LIN {X 0.048,Y -151.819,Z 1203.251,A 0.000,B 0.000,C 90.000,E1 225.162} C_DIS
LIN {X 0.060,Y -150.032,Z 1203.236,A 0.000,B 0.000,C 90.000,E1 222.447} C_DIS
LIN {X -0.026,Y -146.851,Z 1203.211,A 0.000,B 0.000,C 90.000,E1 217.935} C_DIS
LIN {X -0.008,Y -145.434,Z 1203.195,A 0.000,B 0.000,C 90.000,E1 215.185} C_DIS
LIN {X -0.012,Y -142.857,Z 1203.170,A 0.000,B 0.000,C 90.000,E1 210.590} C_DIS
LIN {X 0.040,Y -141.472,Z 1203.149,A 0.000,B 0.000,C 90.000,E1 206.873} C_DIS
LIN {X 0.031,Y -139.379,Z 1203.113,A 0.000,B 0.000,C 90.000,E1 200.375} C_DIS
LIN {X 0.021,Y -138.831,Z 1203.098,A 0.000,B 0.000,C 90.000,E1 197.583} C_DIS
LIN {X -0.051,Y -138.353,Z 1203.056,A 0.000,B 0.000,C 90.000,E1 190.141} C_DIS
LIN {X -0.056,Y -139.527,Z 1203.004,A 0.000,B 0.000,C 90.000,E1 180.802} C_DIS
LIN {X 0.036,Y -141.198,Z 1202.973,A 0.000,B 0.000,C 90.000,E1 175.179} C_DIS
LIN {X -0.005,Y -142.575,Z 1202.958,A 0.000,B 0.000,C 90.000,E1 172.413} C_DIS
LIN {X -0.050,Y -144.865,Z 1202.932,A 0.000,B 0.000,C 90.000,E1 167.813} C_DIS
LIN {X 0.047,Y -147.491,Z 1202.912,A 0.000,B 0.000,C 90.000,E1 164.102} C_DIS
LIN {X -0.019,Y -150.080,Z 1202.891,A 0.000,B 0.000,C 90.000,E1 160.477} C_DIS
LIN {X -0.006,Y -153.430,Z 1202.871,A 0.000,B 0.000,C 90.000,E1 156.847} C_DIS
LIN {X -0.018,Y -156.851,Z 1202.851,A 0.000,B 0.000,C 90.000,E1 153.256} C_DIS
LIN {X 0.053,Y -160.933,Z 1202.832,A 0.000,B 0.000,C 90.000,E1 149.665} C_DIS
LIN {X -0.004,Y -163.056,Z 1202.822,A 0.000,B 0.000,C 90.000,E1 147.916} C_DIS
LIN {X 0.001,Y -167.451,Z 1202.802,A 0.000,B 0.000,C 90.000,E1 144.402} C_DIS
LIN {X -0.090,Y -171.289,Z 1202.788,A 0.000,B 0.000,C 90.000,E1 141.823} C_DIS
LIN {X 0.080,Y -176.182,Z 1202.769,A 0.000,B 0.000,C 90.000,E1 138.324} C_DIS
LIN {X -0.055,Y -180.457,Z 1202.754,A 0.000,B 0.000,C 90.000,E1 135.810} C_DIS
LIN {X -0.079,Y -185.862,Z 1202.736,A 0.000,B 0.000,C 90.000,E1 132.447} C_DIS
LIN {X -0.026,Y -190.485,Z 1202.722,A 0.000,B 0.000,C 90.000,E1 129.930} C_DIS
LIN {X -0.006,Y -196.237,Z 1202.703,A 0.000,B 0.000,C 90.000,E1 126.629} C_DIS
LIN {X 0.003,Y -201.371,Z 1202.689,A 0.000,B 0.000,C 90.000,E1 123.992} C_DIS
LIN {X 0.020,Y -201.579,Z 1202.688,A 0.000,B 0.000,C 90.000,E1 123.865} C_DIS
LIN {X -0.004,Y -311.934,Z 1202.688,A 0.000,B 0.000,C 90.000,E1 123.865} C_DIS
LIN {X -0.100,Y -314.414,Z 1202.688,A 0.000,B 0.000,C 90.000,E1 123.833} C_DIS
LIN {X 0.095,Y -318.650,Z 1202.687,A 0.000,B 0.000,C 90.000,E1 123.579} C_DIS
LIN {X 0.026,Y -321.137,Z 1202.685,A 0.000,B 0.000,C 90.000,E1 123.372} C_DIS
LIN {X -0.050,Y -324.912,Z 1202.683,A 0.000,B 0.000,C 90.000,E1 122.880} C_DIS
LIN {X 0.036,Y -326.560,Z 1202.681,A 0.000,B 0.000,C 90.000,E1 122.546} C_DIS
LIN {X -0.052,Y -333.737,Z 1202.670,A 0.000,B 0.000,C 90.000,E1 120.669} C_DIS
LIN {X 0.128,Y -345.390,Z 1202.655,A 0.000,B 0.000,C 90.000,E1 117.847} C_DIS
LIN {X -0.146,Y -358.479,Z 1202.640,A 0.000,B 0.000,C 90.000,E1 115.155} C_DIS
LIN {X -0.126,Y -371.413,Z 1202.626,A 0.000,B 0.000,C 90.000,E1 112.770} C_DIS
LIN {X -0.068,Y -385.665,Z 1202.613,A 0.000,B 0.000,C 90.000,E1 110.429} C_DIS
LIN {X 0.090,Y -401.333,Z 1202.601,A 0.000,B 0.000,C 90.000,E1 108.127} C_DIS
LIN {X 0.132,Y -418.530,Z 1202.588,A 0.000,B 0.000,C 90.000,E1 105.898} C_DIS
LIN {X -0.161,Y -437.373,Z 1202.576,A 0.000,B 0.000,C 90.000,E1 103.772} C_DIS
LIN {X -0.061,Y -457.365,Z 1202.565,A 0.000,B 0.000,C 90.000,E1 101.715} C_DIS
LIN {X 0.202,Y -470.159,Z 1202.558,A 0.000,B 0.000,C 90.000,E1 100.489} C_DIS
LIN {X -0.210,Y -472.456,Z 1202.557,A 0.000,B 0.000,C 90.000,E1 100.310} C_DIS
LIN {X -0.161,Y -474.191,Z 1202.556,A 0.000,B 0.000,C 90.000,E1 100.074} C_DIS
LIN {X 0.087,Y -475.642,Z 1202.554,A 0.000,B 0.000,C 90.000,E1 99.792} C_DIS
LIN {X -0.053,Y -476.723,Z 1202.553,A 0.000,B 0.000,C 90.000,E1 99.557} C_DIS
LIN {X 0.155,Y -477.992,Z 1202.550,A 0.000,B 0.000,C 90.000,E1 99.029} C_DIS
LIN {X -0.179,Y -478.247,Z 1202.547,A 0.000,B 0.000,C 90.000,E1 98.568} C_DIS
LIN {X -0.032,Y -477.531,Z 1202.545,A 0.000,B 0.000,C 90.000,E1 98.049} C_DIS
LIN {X 0.120,Y -475.728,Z 1202.542,A 0.000,B 0.000,C 90.000,E1 97.530} C_DIS
LIN {X -0.012,Y -474.315,Z 1202.541,A 0.000,B 0.000,C 90.000,E1 97.296} C_DIS
LIN {X 0.182,Y -457.953,Z 1202.528,A 0.000,B 0.000,C 90.000,E1 94.992} C_DIS
LIN {X 0.101,Y -440.459,Z 1202.513,A 0.000,B 0.000,C 90.000,E1 92.407} C_DIS
LIN {X 0.061,Y -422.849,Z 1202.497,A 0.000,B 0.000,C 90.000,E1 89.484} C_DIS
LIN {X 0.074,Y -411.058,Z 1202.485,A 0.000,B 0.000,C 90.000,E1 87.306} C_DIS
LIN {X -0.140,Y -399.438,Z 1202.473,A 0.000,B 0.000,C 90.000,E1 85.122} C_DIS
LIN {X 0.154,Y -389.245,Z 1202.462,A 0.000,B 0.000,C 90.000,E1 83.109} C_DIS
LIN {X -0.068,Y -378.977,Z 1202.451,A 0.000,B 0.000,C 90.000,E1 81.141} C_DIS
LIN {X -0.060,Y -369.917,Z 1202.441,A 0.000,B 0.000,C 90.000,E1 79.398} C_DIS
LIN {X -0.178,Y -358.952,Z 1202.430,A 0.000,B 0.000,C 90.000,E1 77.353} C_DIS
LIN {X -0.028,Y -347.727,Z 1202.418,A 0.000,B 0.000,C 90.000,E1 75.227} C_DIS
LIN {X -0.027,Y -336.543,Z 1202.406,A 0.000,B 0.000,C 90.000,E1 73.087} C_DIS
LIN {X 0.152,Y -322.352,Z 1202.390,A 0.000,B 0.000,C 90.000,E1 70.242} C_DIS
LIN {X 0.074,Y -307.432,Z 1202.373,A 0.000,B 0.000,C 90.000,E1 67.050} C_DIS
LIN {X 0.028,Y -293.601,Z 1202.354,A 0.000,B 0.000,C 90.000,E1 63.768} C_DIS
LIN {X 0.128,Y -281.957,Z 1202.337,A 0.000,B 0.000,C 90.000,E1 60.717} C_DIS
LIN {X -0.128,Y -269.872,Z 1202.318,A 0.000,B 0.000,C 90.000,E1 57.327} C_DIS
LIN {X -0.026,Y -258.643,Z 1202.299,A 0.000,B 0.000,C 90.000,E1 53.783} C_DIS
LIN {X 0.118,Y -250.151,Z 1202.283,A 0.000,B 0.000,C 90.000,E1 50.884} C_DIS
LIN {X -0.016,Y -242.089,Z 1202.267,A 0.000,B 0.000,C 90.000,E1 48.000} C_DIS
LIN {X -0.024,Y -234.378,Z 1202.250,A 0.000,B 0.000,C 90.000,E1 45.040} C_DIS
LIN {X -0.021,Y -225.204,Z 1202.229,A 0.000,B 0.000,C 90.000,E1 41.272} C_DIS
LIN {X 0.094,Y -218.537,Z 1202.212,A 0.000,B 0.000,C 90.000,E1 38.177} C_DIS
LIN {X -0.043,Y -212.560,Z 1202.195,A 0.000,B 0.000,C 90.000,E1 35.105} C_DIS
LIN {X 0.079,Y -205.966,Z 1202.173,A 0.000,B 0.000,C 90.000,E1 31.131} C_DIS
LIN {X 0.100,Y -200.208,Z 1202.151,A 0.000,B 0.000,C 90.000,E1 27.129} C_DIS
LIN {X -0.063,Y -195.149,Z 1202.128,A 0.000,B 0.000,C 90.000,E1 23.131} C_DIS
LIN {X -0.033,Y -190.918,Z 1202.106,A 0.000,B 0.000,C 90.000,E1 19.033} C_DIS
LIN {X 0.012,Y -186.961,Z 1202.078,A 0.000,B 0.000,C 90.000,E1 14.064} C_DIS
LIN {X 0.052,Y -184.087,Z 1202.046,A 0.000,B 0.000,C 90.000,E1 8.219} C_DIS
LIN {X 0.056,Y -184.995,Z 1201.969,A 0.000,B 0.000,C 90.000,E1 354.489} C_DIS
LIN {X -0.023,Y -187.980,Z 1201.942,A 0.000,B 0.000,C 90.000,E1 349.511} C_DIS
LIN {X 0.033,Y -191.482,Z 1201.919,A 0.000,B 0.000,C 90.000,E1 345.353} C_DIS
LIN {X -0.066,Y -195.946,Z 1201.896,A 0.000,B 0.000,C 90.000,E1 341.275} C_DIS
LIN {X 0.047,Y -201.140,Z 1201.873,A 0.000,B 0.000,C 90.000,E1 337.177} C_DIS
LIN {X -0.017,Y -207.027,Z 1201.851,A 0.000,B 0.000,C 90.000,E1 333.179} C_DIS
LIN {X 0.020,Y -213.376,Z 1201.829,A 0.000,B 0.000,C 90.000,E1 329.203} C_DIS
LIN {X -0.041,Y -220.263,Z 1201.807,A 0.000,B 0.000,C 90.000,E1 325.308} C_DIS
LIN {X -0.046,Y -227.871,Z 1201.786,A 0.000,B 0.000,C 90.000,E1 321.457} C_DIS
LIN {X 0.010,Y -234.629,Z 1201.769,A 0.000,B 0.000,C 90.000,E1 318.405} C_DIS
LIN {X 0.027,Y -242.403,Z 1201.752,A 0.000,B 0.000,C 90.000,E1 315.405} C_DIS
LIN {X -0.071,Y -250.248,Z 1201.738,A 0.000,B 0.000,C 90.000,E1 312.852} C_DIS
LIN {X 0.053,Y -260.364,Z 1201.722,A 0.000,B 0.000,C 90.000,E1 309.930} C_DIS
LIN {X 0.054,Y -272.944,Z 1201.704,A 0.000,B 0.000,C 90.000,E1 306.744} C_DIS
LIN {X 0.028,Y -283.932,Z 1201.691,A 0.000,B 0.000,C 90.000,E1 304.326} C_DIS
LIN {X -0.001,Y -295.991,Z 1201.677,A 0.000,B 0.000,C 90.000,E1 301.957} C_DIS
LIN {X 0.067,Y -307.506,Z 1201.667,A 0.000,B 0.000,C 90.000,E1 299.951} C_DIS
LIN {X -0.132,Y -318.187,Z 1201.657,A 0.000,B 0.000,C 90.000,E1 298.359} C_DIS
LIN {X 0.012,Y -327.551,Z 1201.650,A 0.000,B 0.000,C 90.000,E1 297.052} C_DIS
LIN {X 0.102,Y -337.663,Z 1201.643,A 0.000,B 0.000,C 90.000,E1 295.796} C_DIS
LIN {X 0.001,Y -350.670,Z 1201.635,A 0.000,B 0.000,C 90.000,E1 294.335} C_DIS
LIN {X 0.036,Y -369.290,Z 1201.624,A 0.000,B 0.000,C 90.000,E1 292.333} C_DIS
LIN {X 0.131,Y -388.068,Z 1201.614,A 0.000,B 0.000,C 90.000,E1 290.429} C_DIS
LIN {X 0.065,Y -398.725,Z 1201.608,A 0.000,B 0.000,C 90.000,E1 289.396} C_DIS
LIN {X -0.053,Y -411.786,Z 1201.601,A 0.000,B 0.000,C 90.000,E1 288.109} C_DIS
LIN {X -0.193,Y -421.737,Z 1201.595,A 0.000,B 0.000,C 90.000,E1 287.094} C_DIS
LIN {X 0.081,Y -428.965,Z 1201.590,A 0.000,B 0.000,C 90.000,E1 286.260} C_DIS
LIN {X -0.123,Y -435.805,Z 1201.586,A 0.000,B 0.000,C 90.000,E1 285.481} C_DIS
LIN {X 0.032,Y -442.017,Z 1201.581,A 0.000,B 0.000,C 90.000,E1 284.662} C_DIS
LIN {X -0.064,Y -447.642,Z 1201.577,A 0.000,B 0.000,C 90.000,E1 283.883} C_DIS
LIN {X 0.211,Y -452.582,Z 1201.573,A 0.000,B 0.000,C 90.000,E1 283.063} C_DIS
LIN {X 0.098,Y -456.793,Z 1201.568,A 0.000,B 0.000,C 90.000,E1 282.299} C_DIS
LIN {X 0.016,Y -460.399,Z 1201.564,A 0.000,B 0.000,C 90.000,E1 281.535} C_DIS
LIN {X 0.129,Y -462.357,Z 1201.561,A 0.000,B 0.000,C 90.000,E1 281.007} C_DIS
LIN {X 0.163,Y -464.083,Z 1201.558,A 0.000,B 0.000,C 90.000,E1 280.489} C_DIS
LIN {X -0.164,Y -465.496,Z 1201.556,A 0.000,B 0.000,C 90.000,E1 280.018} C_DIS
LIN {X -0.104,Y -466.634,Z 1201.553,A 0.000,B 0.000,C 90.000,E1 279.500} C_DIS
LIN {X 0.120,Y -468.298,Z 1201.547,A 0.000,B 0.000,C 90.000,E1 278.454} C_DIS
LIN {X 0.207,Y -468.819,Z 1201.544,A 0.000,B 0.000,C 90.000,E1 277.936} C_DIS
LIN {X -0.103,Y -469.122,Z 1201.541,A 0.000,B 0.000,C 90.000,E1 277.466} C_DIS
LIN {X -0.010,Y -469.099,Z 1201.539,A 0.000,B 0.000,C 90.000,E1 276.947} C_DIS
LIN {X 0.086,Y -468.688,Z 1201.536,A 0.000,B 0.000,C 90.000,E1 276.429} C_DIS
LIN {X 0.181,Y -467.860,Z 1201.533,A 0.000,B 0.000,C 90.000,E1 275.910} C_DIS
LIN {X -0.192,Y -466.569,Z 1201.530,A 0.000,B 0.000,C 90.000,E1 275.448} C_DIS
LIN {X -0.145,Y -464.814,Z 1201.527,A 0.000,B 0.000,C 90.000,E1 274.935} C_DIS
LIN {X -0.064,Y -462.513,Z 1201.525,A 0.000,B 0.000,C 90.000,E1 274.416} C_DIS
LIN {X -0.003,Y -459.600,Z 1201.522,A 0.000,B 0.000,C 90.000,E1 273.898} C_DIS
LIN {X -0.224,Y -457.878,Z 1201.520,A 0.000,B 0.000,C 90.000,E1 273.669} C_DIS
LIN {X -0.188,Y -453.649,Z 1201.517,A 0.000,B 0.000,C 90.000,E1 273.151} C_DIS
LIN {X 0.037,Y -451.115,Z 1201.516,A 0.000,B 0.000,C 90.000,E1 272.865} C_DIS
LIN {X -0.156,Y -448.310,Z 1201.515,A 0.000,B 0.000,C 90.000,E1 272.636} C_DIS
LIN {X -0.210,Y -442.028,Z 1201.512,A 0.000,B 0.000,C 90.000,E1 272.178} C_DIS
LIN {X -0.055,Y -435.183,Z 1201.510,A 0.000,B 0.000,C 90.000,E1 271.776} C_DIS
LIN {X 0.204,Y -428.018,Z 1201.508,A 0.000,B 0.000,C 90.000,E1 271.432} C_DIS
LIN {X 0.005,Y -421.056,Z 1201.507,A 0.000,B 0.000,C 90.000,E1 271.203} C_DIS
LIN {X 0.166,Y -410.827,Z 1201.505,A 0.000,B 0.000,C 90.000,E1 270.859} C_DIS
LIN {X -0.140,Y -400.798,Z 1201.503,A 0.000,B 0.000,C 90.000,E1 270.630} C_DIS
LIN {X -0.039,Y -393.335,Z 1201.503,A 0.000,B 0.000,C 90.000,E1 270.458} C_DIS
LIN {X -0.139,Y -381.231,Z 1201.501,A 0.000,B 0.000,C 90.000,E1 270.286} C_DIS
LIN {X 0.134,Y -373.463,Z 1201.501,A 0.000,B 0.000,C 90.000,E1 270.172} C_DIS
LIN {X -0.073,Y -366.137,Z 1201.501,A 0.000,B 0.000,C 90.000,E1 270.172} C_DIS
LIN {X -0.061,Y -181.578,Z 1201.501,A 0.000,B 0.000,C 90.000,E1 270.172} C_DIS
LIN {X -0.033,Y -180.873,Z 1201.473,A 0.000,B 0.000,C 90.000,E1 265.065} C_DIS
LIN {X 0.024,Y -178.990,Z 1201.444,A 0.000,B 0.000,C 90.000,E1 259.982} C_DIS
LIN {X 0.035,Y -177.975,Z 1201.435,A 0.000,B 0.000,C 90.000,E1 258.285} C_DIS
LIN {X 0.054,Y -175.618,Z 1201.411,A 0.000,B 0.000,C 90.000,E1 254.031} C_DIS
LIN {X 0.065,Y -172.340,Z 1201.388,A 0.000,B 0.000,C 90.000,E1 249.752} C_DIS
LIN {X 0.044,Y -171.816,Z 1201.383,A 0.000,B 0.000,C 90.000,E1 248.901} C_DIS
LIN {X 0.051,Y -170.282,Z 1201.373,A 0.000,B 0.000,C 90.000,E1 247.177} C_DIS
LIN {X -0.013,Y -166.822,Z 1201.349,A 0.000,B 0.000,C 90.000,E1 242.871} C_DIS
LIN {X -0.095,Y -162.804,Z 1201.325,A 0.000,B 0.000,C 90.000,E1 238.535} C_DIS
LIN {X -0.031,Y -161.490,Z 1201.315,A 0.000,B 0.000,C 90.000,E1 236.755} C_DIS
LIN {X 0.019,Y -157.487,Z 1201.291,A 0.000,B 0.000,C 90.000,E1 232.316} C_DIS
LIN {X -0.043,Y -155.505,Z 1201.276,A 0.000,B 0.000,C 90.000,E1 229.666} C_DIS
LIN {X 0.008,Y -151.808,Z 1201.251,A 0.000,B 0.000,C 90.000,E1 225.162} C_DIS
LIN {X 0.020,Y -150.019,Z 1201.236,A 0.000,B 0.000,C 90.000,E1 222.447} C_DIS
LIN {X 0.051,Y -146.842,Z 1201.211,A 0.000,B 0.000,C 90.000,E1 217.890} C_DIS
LIN {X -0.047,Y -145.424,Z 1201.195,A 0.000,B 0.000,C 90.000,E1 215.185} C_DIS
LIN {X -0.051,Y -142.850,Z 1201.170,A 0.000,B 0.000,C 90.000,E1 210.590} C_DIS
LIN {X 0.002,Y -141.465,Z 1201.149,A 0.000,B 0.000,C 90.000,E1 206.873} C_DIS
LIN {X -0.007,Y -139.377,Z 1201.113,A 0.000,B 0.000,C 90.000,E1 200.375} C_DIS
LIN {X -0.017,Y -138.828,Z 1201.098,A 0.000,B 0.000,C 90.000,E1 197.583} C_DIS
LIN {X 0.047,Y -138.353,Z 1201.056,A 0.000,B 0.000,C 90.000,E1 190.084} C_DIS
LIN {X 0.045,Y -139.529,Z 1201.004,A 0.000,B 0.000,C 90.000,E1 180.745} C_DIS
LIN {X -0.002,Y -141.205,Z 1200.973,A 0.000,B 0.000,C 90.000,E1 175.179} C_DIS
LIN {X -0.043,Y -142.580,Z 1200.958,A 0.000,B 0.000,C 90.000,E1 172.413} C_DIS
LIN {X 0.053,Y -144.875,Z 1200.932,A 0.000,B 0.000,C 90.000,E1 167.757} C_DIS
LIN {X 0.007,Y -147.501,Z 1200.912,A 0.000,B 0.000,C 90.000,E1 164.102} C_DIS
LIN {X 0.082,Y -150.092,Z 1200.891,A 0.000,B 0.000,C 90.000,E1 160.423} C_DIS
LIN {X -0.046,Y -153.447,Z 1200.871,A 0.000,B 0.000,C 90.000,E1 156.847} C_DIS
LIN {X -0.053,Y -157.809,Z 1200.846,A 0.000,B 0.000,C 90.000,E1 152.359} C_DIS
LIN {X -0.020,Y -162.092,Z 1200.827,A 0.000,B 0.000,C 90.000,E1 148.791} C_DIS
LIN {X 0.004,Y -166.291,Z 1200.807,A 0.000,B 0.000,C 90.000,E1 145.261} C_DIS
LIN {X 0.001,Y -171.308,Z 1200.788,A 0.000,B 0.000,C 90.000,E1 141.778} C_DIS
LIN {X 0.036,Y -176.205,Z 1200.769,A 0.000,B 0.000,C 90.000,E1 138.324} C_DIS
LIN {X -0.099,Y -180.482,Z 1200.754,A 0.000,B 0.000,C 90.000,E1 135.810} C_DIS
LIN {X 0.012,Y -185.886,Z 1200.736,A 0.000,B 0.000,C 90.000,E1 132.405} C_DIS
LIN {X -0.073,Y -190.512,Z 1200.722,A 0.000,B 0.000,C 90.000,E1 129.930} C_DIS
LIN {X 0.105,Y -196.264,Z 1200.703,A 0.000,B 0.000,C 90.000,E1 126.583} C_DIS
LIN {X -0.044,Y -201.393,Z 1200.689,A 0.000,B 0.000,C 90.000,E1 123.992} C_DIS
LIN {X -0.027,Y -201.603,Z 1200.688,A 0.000,B 0.000,C 90.000,E1 123.865} C_DIS
LIN {X -0.078,Y -311.928,Z 1200.688,A 0.000,B 0.000,C 90.000,E1 123.865} C_DIS
LIN {X 0.088,Y -314.438,Z 1200.688,A 0.000,B 0.000,C 90.000,E1 123.785} C_DIS
LIN {X 0.019,Y -318.680,Z 1200.687,A 0.000,B 0.000,C 90.000,E1 123.579} C_DIS
LIN {X -0.050,Y -321.168,Z 1200.685,A 0.000,B 0.000,C 90.000,E1 123.372} C_DIS
LIN {X -0.126,Y -324.942,Z 1200.682,A 0.000,B 0.000,C 90.000,E1 122.880} C_DIS
LIN {X -0.039,Y -326.589,Z 1200.681,A 0.000,B 0.000,C 90.000,E1 122.546} C_DIS
LIN {X -0.129,Y -333.767,Z 1200.670,A 0.000,B 0.000,C 90.000,E1 120.669} C_DIS
LIN {X 0.050,Y -345.426,Z 1200.655,A 0.000,B 0.000,C 90.000,E1 117.847} C_DIS
LIN {X -0.227,Y -358.521,Z 1200.640,A 0.000,B 0.000,C 90.000,E1 115.155} C_DIS
LIN {X -0.209,Y -371.463,Z 1200.626,A 0.000,B 0.000,C 90.000,E1 112.770} C_DIS
LIN {X -0.153,Y -385.722,Z 1200.613,A 0.000,B 0.000,C 90.000,E1 110.429} C_DIS
LIN {X 0.004,Y -401.397,Z 1200.601,A 0.000,B 0.000,C 90.000,E1 108.127} C_DIS
LIN {X 0.043,Y -418.602,Z 1200.588,A 0.000,B 0.000,C 90.000,E1 105.898} C_DIS
LIN {X -0.251,Y -437.454,Z 1200.576,A 0.000,B 0.000,C 90.000,E1 103.772} C_DIS
LIN {X -0.148,Y -457.449,Z 1200.565,A 0.000,B 0.000,C 90.000,E1 101.715} C_DIS
LIN {X 0.117,Y -470.245,Z 1200.558,A 0.000,B 0.000,C 90.000,E1 100.489} C_DIS
LIN {X 0.170,Y -472.498,Z 1200.557,A 0.000,B 0.000,C 90.000,E1 100.254} C_DIS
LIN {X 0.221,Y -474.200,Z 1200.556,A 0.000,B 0.000,C 90.000,E1 100.018} C_DIS
LIN {X 0.001,Y -475.625,Z 1200.554,A 0.000,B 0.000,C 90.000,E1 99.792} C_DIS
LIN {X -0.137,Y -476.684,Z 1200.553,A 0.000,B 0.000,C 90.000,E1 99.557} C_DIS
LIN {X 0.069,Y -477.919,Z 1200.550,A 0.000,B 0.000,C 90.000,E1 99.029} C_DIS
LIN {X 0.208,Y -478.143,Z 1200.547,A 0.000,B 0.000,C 90.000,E1 98.511} C_DIS
LIN {X -0.117,Y -477.395,Z 1200.545,A 0.000,B 0.000,C 90.000,E1 98.049} C_DIS
LIN {X 0.033,Y -475.555,Z 1200.542,A 0.000,B 0.000,C 90.000,E1 97.530} C_DIS
LIN {X -0.099,Y -474.116,Z 1200.540,A 0.000,B 0.000,C 90.000,E1 97.296} C_DIS
LIN {X 0.092,Y -457.754,Z 1200.528,A 0.000,B 0.000,C 90.000,E1 94.992} C_DIS
LIN {X 0.011,Y -440.246,Z 1200.513,A 0.000,B 0.000,C 90.000,E1 92.407} C_DIS
LIN {X -0.032,Y -422.644,Z 1200.497,A 0.000,B 0.000,C 90.000,E1 89.484} C_DIS
LIN {X -0.022,Y -410.862,Z 1200.485,A 0.000,B 0.000,C 90.000,E1 87.306} C_DIS
LIN {X 0.160,Y -399.222,Z 1200.473,A 0.000,B 0.000,C 90.000,E1 85.065} C_DIS
LIN {X 0.055,Y -389.034,Z 1200.462,A 0.000,B 0.000,C 90.000,E1 83.109} C_DIS
LIN {X -0.169,Y -378.779,Z 1200.451,A 0.000,B 0.000,C 90.000,E1 81.141} C_DIS
LIN {X -0.160,Y -371.241,Z 1200.443,A 0.000,B 0.000,C 90.000,E1 79.690} C_DIS
LIN {X 0.130,Y -361.903,Z 1200.433,A 0.000,B 0.000,C 90.000,E1 77.881} C_DIS
LIN {X -0.031,Y -352.343,Z 1200.423,A 0.000,B 0.000,C 90.000,E1 76.117} C_DIS
LIN {X -0.028,Y -339.516,Z 1200.409,A 0.000,B 0.000,C 90.000,E1 73.685} C_DIS
LIN {X -0.142,Y -326.773,Z 1200.396,A 0.000,B 0.000,C 90.000,E1 71.221} C_DIS
LIN {X -0.075,Y -311.600,Z 1200.378,A 0.000,B 0.000,C 90.000,E1 68.028} C_DIS
LIN {X 0.044,Y -296.090,Z 1200.358,A 0.000,B 0.000,C 90.000,E1 64.409} C_DIS
LIN {X 0.046,Y -283.018,Z 1200.339,A 0.000,B 0.000,C 90.000,E1 61.051} C_DIS
LIN {X -0.177,Y -270.840,Z 1200.320,A 0.000,B 0.000,C 90.000,E1 57.661} C_DIS
LIN {X -0.088,Y -260.598,Z 1200.303,A 0.000,B 0.000,C 90.000,E1 54.482} C_DIS
LIN {X -0.052,Y -251.980,Z 1200.287,A 0.000,B 0.000,C 90.000,E1 51.618} C_DIS
LIN {X 0.045,Y -241.790,Z 1200.266,A 0.000,B 0.000,C 90.000,E1 47.957} C_DIS
LIN {X 0.018,Y -234.061,Z 1200.250,A 0.000,B 0.000,C 90.000,E1 45.000} C_DIS
LIN {X 0.020,Y -224.883,Z 1200.229,A 0.000,B 0.000,C 90.000,E1 41.229} C_DIS
LIN {X -0.038,Y -218.246,Z 1200.212,A 0.000,B 0.000,C 90.000,E1 38.177} C_DIS
LIN {X -0.021,Y -210.917,Z 1200.190,A 0.000,B 0.000,C 90.000,E1 34.278} C_DIS
LIN {X -0.057,Y -204.484,Z 1200.168,A 0.000,B 0.000,C 90.000,E1 30.335} C_DIS
LIN {X 0.006,Y -198.854,Z 1200.146,A 0.000,B 0.000,C 90.000,E1 26.309} C_DIS
LIN {X -0.018,Y -193.929,Z 1200.124,A 0.000,B 0.000,C 90.000,E1 22.259} C_DIS
LIN {X -0.091,Y -189.862,Z 1200.101,A 0.000,B 0.000,C 90.000,E1 18.181} C_DIS
LIN {X 0.038,Y -186.108,Z 1200.073,A 0.000,B 0.000,C 90.000,E1 13.175} C_DIS
LIN {X -0.026,Y -183.490,Z 1200.041,A 0.000,B 0.000,C 90.000,E1 7.352} C_DIS
LIN {X 0.044,Y -184.640,Z 1199.969,A 0.000,B 0.000,C 90.000,E1 354.489} C_DIS
LIN {X -0.049,Y -187.652,Z 1199.942,A 0.000,B 0.000,C 90.000,E1 349.511} C_DIS
LIN {X 0.045,Y -191.145,Z 1199.919,A 0.000,B 0.000,C 90.000,E1 345.338} C_DIS
LIN {X 0.071,Y -195.623,Z 1199.896,A 0.000,B 0.000,C 90.000,E1 341.221} C_DIS
LIN {X -0.013,Y -200.824,Z 1199.873,A 0.000,B 0.000,C 90.000,E1 337.177} C_DIS
LIN {X 0.096,Y -206.697,Z 1199.851,A 0.000,B 0.000,C 90.000,E1 333.127} C_DIS
LIN {X -0.064,Y -213.098,Z 1199.829,A 0.000,B 0.000,C 90.000,E1 329.203} C_DIS
LIN {X 0.044,Y -219.987,Z 1199.807,A 0.000,B 0.000,C 90.000,E1 325.261} C_DIS
LIN {X 0.025,Y -227.630,Z 1199.786,A 0.000,B 0.000,C 90.000,E1 321.412} C_DIS
LIN {X -0.107,Y -234.420,Z 1199.769,A 0.000,B 0.000,C 90.000,E1 318.405} C_DIS
LIN {X 0.108,Y -241.216,Z 1199.754,A 0.000,B 0.000,C 90.000,E1 315.729} C_DIS
LIN {X -0.017,Y -248.968,Z 1199.740,A 0.000,B 0.000,C 90.000,E1 313.176} C_DIS
LIN {X 0.079,Y -258.991,Z 1199.724,A 0.000,B 0.000,C 90.000,E1 310.253} C_DIS
LIN {X 0.000,Y -271.454,Z 1199.706,A 0.000,B 0.000,C 90.000,E1 307.076} C_DIS
LIN {X 0.056,Y -280.695,Z 1199.694,A 0.000,B 0.000,C 90.000,E1 304.978} C_DIS
LIN {X 0.016,Y -294.242,Z 1199.679,A 0.000,B 0.000,C 90.000,E1 302.260} C_DIS
LIN {X 0.041,Y -305.597,Z 1199.668,A 0.000,B 0.000,C 90.000,E1 300.256} C_DIS
LIN {X 0.077,Y -316.097,Z 1199.659,A 0.000,B 0.000,C 90.000,E1 298.615} C_DIS
LIN {X 0.050,Y -325.197,Z 1199.652,A 0.000,B 0.000,C 90.000,E1 297.334} C_DIS
LIN {X -0.157,Y -335.220,Z 1199.645,A 0.000,B 0.000,C 90.000,E1 296.104} C_DIS
LIN {X -0.068,Y -348.527,Z 1199.636,A 0.000,B 0.000,C 90.000,E1 294.567} C_DIS
LIN {X -0.022,Y -369.661,Z 1199.624,A 0.000,B 0.000,C 90.000,E1 292.280} C_DIS
LIN {X 0.099,Y -388.519,Z 1199.613,A 0.000,B 0.000,C 90.000,E1 290.375} C_DIS
LIN {X 0.196,Y -399.152,Z 1199.608,A 0.000,B 0.000,C 90.000,E1 289.322} C_DIS
LIN {X -0.049,Y -412.269,Z 1199.600,A 0.000,B 0.000,C 90.000,E1 288.055} C_DIS
LIN {X 0.096,Y -422.356,Z 1199.594,A 0.000,B 0.000,C 90.000,E1 286.985} C_DIS
LIN {X -0.114,Y -429.647,Z 1199.590,A 0.000,B 0.000,C 90.000,E1 286.205} C_DIS
LIN {X 0.105,Y -436.435,Z 1199.585,A 0.000,B 0.000,C 90.000,E1 285.371} C_DIS
LIN {X -0.043,Y -442.604,Z 1199.581,A 0.000,B 0.000,C 90.000,E1 284.592} C_DIS
LIN {X 0.188,Y -448.152,Z 1199.577,A 0.000,B 0.000,C 90.000,E1 283.772} C_DIS
LIN {X 0.033,Y -453.054,Z 1199.572,A 0.000,B 0.000,C 90.000,E1 283.008} C_DIS
LIN {X -0.076,Y -457.216,Z 1199.568,A 0.000,B 0.000,C 90.000,E1 282.243} C_DIS
LIN {X -0.156,Y -460.722,Z 1199.564,A 0.000,B 0.000,C 90.000,E1 281.478} C_DIS
LIN {X -0.041,Y -462.667,Z 1199.561,A 0.000,B 0.000,C 90.000,E1 280.950} C_DIS
LIN {X -0.004,Y -464.344,Z 1199.558,A 0.000,B 0.000,C 90.000,E1 280.433} C_DIS
LIN {X 0.129,Y -465.691,Z 1199.555,A 0.000,B 0.000,C 90.000,E1 279.905} C_DIS
LIN {X -0.191,Y -466.765,Z 1199.552,A 0.000,B 0.000,C 90.000,E1 279.434} C_DIS
LIN {X -0.040,Y -468.394,Z 1199.547,A 0.000,B 0.000,C 90.000,E1 278.398} C_DIS
LIN {X 0.112,Y -468.937,Z 1199.544,A 0.000,B 0.000,C 90.000,E1 277.871} C_DIS
LIN {X 0.203,Y -469.252,Z 1199.541,A 0.000,B 0.000,C 90.000,E1 277.352} C_DIS
LIN {X -0.168,Y -469.208,Z 1199.538,A 0.000,B 0.000,C 90.000,E1 276.891} C_DIS
LIN {X -0.071,Y -468.781,Z 1199.535,A 0.000,B 0.000,C 90.000,E1 276.372} C_DIS
LIN {X 0.027,Y -467.890,Z 1199.533,A 0.000,B 0.000,C 90.000,E1 275.853} C_DIS
LIN {X 0.120,Y -466.521,Z 1199.530,A 0.000,B 0.000,C 90.000,E1 275.334} C_DIS
LIN {X 0.166,Y -464.706,Z 1199.527,A 0.000,B 0.000,C 90.000,E1 274.821} C_DIS
LIN {X -0.215,Y -462.350,Z 1199.524,A 0.000,B 0.000,C 90.000,E1 274.359} C_DIS
LIN {X -0.153,Y -459.324,Z 1199.521,A 0.000,B 0.000,C 90.000,E1 273.841} C_DIS
LIN {X -0.137,Y -455.515,Z 1199.518,A 0.000,B 0.000,C 90.000,E1 273.326} C_DIS
LIN {X 0.114,Y -453.212,Z 1199.517,A 0.000,B 0.000,C 90.000,E1 273.037} C_DIS
LIN {X -0.114,Y -450.597,Z 1199.516,A 0.000,B 0.000,C 90.000,E1 272.808} C_DIS
LIN {X 0.178,Y -447.753,Z 1199.514,A 0.000,B 0.000,C 90.000,E1 272.522} C_DIS
LIN {X 0.186,Y -441.359,Z 1199.512,A 0.000,B 0.000,C 90.000,E1 272.064} C_DIS
LIN {X -0.033,Y -434.384,Z 1199.510,A 0.000,B 0.000,C 90.000,E1 271.718} C_DIS
LIN {X -0.148,Y -427.347,Z 1199.508,A 0.000,B 0.000,C 90.000,E1 271.432} C_DIS
LIN {X 0.114,Y -420.347,Z 1199.506,A 0.000,B 0.000,C 90.000,E1 271.146} C_DIS
LIN {X 0.048,Y -407.056,Z 1199.504,A 0.000,B 0.000,C 90.000,E1 270.745} C_DIS
LIN {X -0.157,Y -396.289,Z 1199.503,A 0.000,B 0.000,C 90.000,E1 270.516} C_DIS
LIN {X 0.064,Y -388.525,Z 1199.502,A 0.000,B 0.000,C 90.000,E1 270.344} C_DIS
LIN {X 0.065,Y -380.202,Z 1199.501,A 0.000,B 0.000,C 90.000,E1 270.229} C_DIS
LIN {X -0.021,Y -371.904,Z 1199.501,A 0.000,B 0.000,C 90.000,E1 270.172} C_DIS
LIN {X -0.170,Y -365.589,Z 1199.501,A 0.000,B 0.000,C 90.000,E1 270.172} C_DIS
LIN {X 0.075,Y -181.577,Z 1199.501,A 0.000,B 0.000,C 90.000,E1 270.115} C_DIS
LIN {X 0.086,Y -180.870,Z 1199.472,A 0.000,B 0.000,C 90.000,E1 265.008} C_DIS
LIN {X -0.037,Y -178.985,Z 1199.444,A 0.000,B 0.000,C 90.000,E1 259.982} C_DIS
LIN {X -0.025,Y -177.962,Z 1199.435,A 0.000,B 0.000,C 90.000,E1 258.285} C_DIS
LIN {X -0.006,Y -175.604,Z 1199.411,A 0.000,B 0.000,C 90.000,E1 254.031} C_DIS
LIN {X 0.007,Y -172.327,Z 1199.388,A 0.000,B 0.000,C 90.000,E1 249.752} C_DIS
LIN {X -0.015,Y -171.804,Z 1199.383,A 0.000,B 0.000,C 90.000,E1 248.901} C_DIS
LIN {X -0.007,Y -170.264,Z 1199.373,A 0.000,B 0.000,C 90.000,E1 247.177} C_DIS
LIN {X -0.070,Y -166.806,Z 1199.349,A 0.000,B 0.000,C 90.000,E1 242.871} C_DIS
LIN {X 0.072,Y -162.788,Z 1199.325,A 0.000,B 0.000,C 90.000,E1 238.456} C_DIS
LIN {X 0.047,Y -161.476,Z 1199.315,A 0.000,B 0.000,C 90.000,E1 236.707} C_DIS
LIN {X -0.036,Y -157.472,Z 1199.291,A 0.000,B 0.000,C 90.000,E1 232.316} C_DIS
LIN {X 0.020,Y -155.486,Z 1199.276,A 0.000,B 0.000,C 90.000,E1 229.622} C_DIS
LIN {X -0.047,Y -151.794,Z 1199.251,A 0.000,B 0.000,C 90.000,E1 225.162} C_DIS
LIN {X -0.034,Y -150.003,Z 1199.236,A 0.000,B 0.000,C 90.000,E1 222.447} C_DIS
LIN {X -0.003,Y -146.830,Z 1199.210,A 0.000,B 0.000,C 90.000,E1 217.890} C_DIS
LIN {X -0.016,Y -145.411,Z 1199.195,A 0.000,B 0.000,C 90.000,E1 215.152} C_DIS
LIN {X 0.020,Y -142.841,Z 1199.170,A 0.000,B 0.000,C 90.000,E1 210.541} C_DIS
LIN {X -0.050,Y -141.455,Z 1199.149,A 0.000,B 0.000,C 90.000,E1 206.873} C_DIS
LIN {X -0.010,Y -139.372,Z 1199.113,A 0.000,B 0.000,C 90.000,E1 200.355} C_DIS
LIN {X -0.068,Y -138.822,Z 1199.098,A 0.000,B 0.000,C 90.000,E1 197.583} C_DIS
LIN {X 0.021,Y -138.353,Z 1199.056,A 0.000,B 0.000,C 90.000,E1 190.074} C_DIS
LIN {X -0.007,Y -139.533,Z 1199.004,A 0.000,B 0.000,C 90.000,E1 180.745} C_DIS
LIN {X -0.054,Y -141.214,Z 1198.973,A 0.000,B 0.000,C 90.000,E1 175.179} C_DIS
LIN {X 0.046,Y -142.588,Z 1198.958,A 0.000,B 0.000,C 90.000,E1 172.356} C_DIS
LIN {X 0.000,Y -144.887,Z 1198.932,A 0.000,B 0.000,C 90.000,E1 167.757} C_DIS
LIN {X -0.046,Y -147.515,Z 1198.912,A 0.000,B 0.000,C 90.000,E1 164.102} C_DIS
LIN {X 0.027,Y -150.109,Z 1198.891,A 0.000,B 0.000,C 90.000,E1 160.423} C_DIS
LIN {X 0.040,Y -153.468,Z 1198.871,A 0.000,B 0.000,C 90.000,E1 156.794} C_DIS
LIN {X 0.031,Y -157.831,Z 1198.846,A 0.000,B 0.000,C 90.000,E1 152.308} C_DIS
LIN {X 0.061,Y -162.115,Z 1198.826,A 0.000,B 0.000,C 90.000,E1 148.742} C_DIS
LIN {X -0.054,Y -166.317,Z 1198.807,A 0.000,B 0.000,C 90.000,E1 145.261} C_DIS
LIN {X 0.048,Y -171.335,Z 1198.788,A 0.000,B 0.000,C 90.000,E1 141.743} C_DIS
LIN {X -0.024,Y -176.236,Z 1198.768,A 0.000,B 0.000,C 90.000,E1 138.324} C_DIS
LIN {X 0.095,Y -180.516,Z 1198.754,A 0.000,B 0.000,C 90.000,E1 135.729} C_DIS
LIN {X 0.075,Y -185.919,Z 1198.735,A 0.000,B 0.000,C 90.000,E1 132.366} C_DIS
LIN {X 0.011,Y -190.548,Z 1198.722,A 0.000,B 0.000,C 90.000,E1 129.886} C_DIS
LIN {X 0.042,Y -196.299,Z 1198.703,A 0.000,B 0.000,C 90.000,E1 126.583} C_DIS
LIN {X -0.109,Y -201.425,Z 1198.689,A 0.000,B 0.000,C 90.000,E1 123.992} C_DIS
LIN {X 0.000,Y -201.590,Z 1198.688,A 0.000,B 0.000,C 90.000,E1 123.865} C_DIS
LIN {X -0.048,Y -311.734,Z 1198.688,A 0.000,B 0.000,C 90.000,E1 123.865} C_DIS
LIN {X 0.032,Y -313.074,Z 1198.688,A 0.000,B 0.000,C 90.000,E1 123.833} C_DIS
LIN {X 0.072,Y -318.570,Z 1198.687,A 0.000,B 0.000,C 90.000,E1 123.579} C_DIS
LIN {X -0.153,Y -321.346,Z 1198.685,A 0.000,B 0.000,C 90.000,E1 123.372} C_DIS
LIN {X 0.019,Y -325.060,Z 1198.682,A 0.000,B 0.000,C 90.000,E1 122.832} C_DIS
LIN {X -0.167,Y -326.673,Z 1198.681,A 0.000,B 0.000,C 90.000,E1 122.546} C_DIS
LIN {X 0.087,Y -341.457,Z 1198.660,A 0.000,B 0.000,C 90.000,E1 118.743} C_DIS
LIN {X 0.167,Y -354.075,Z 1198.644,A 0.000,B 0.000,C 90.000,E1 115.976} C_DIS
LIN {X -0.173,Y -368.203,Z 1198.630,A 0.000,B 0.000,C 90.000,E1 113.334} C_DIS
LIN {X -0.058,Y -382.135,Z 1198.616,A 0.000,B 0.000,C 90.000,E1 110.972} C_DIS
LIN {X 0.006,Y -397.460,Z 1198.604,A 0.000,B 0.000,C 90.000,E1 108.671} C_DIS
LIN {X -0.049,Y -414.285,Z 1198.591,A 0.000,B 0.000,C 90.000,E1 106.441} C_DIS
LIN {X 0.077,Y -432.731,Z 1198.579,A 0.000,B 0.000,C 90.000,E1 104.245} C_DIS
LIN {X -0.020,Y -452.551,Z 1198.568,A 0.000,B 0.000,C 90.000,E1 102.175} C_DIS
LIN {X -0.023,Y -470.405,Z 1198.558,A 0.000,B 0.000,C 90.000,E1 100.489} C_DIS
LIN {X 0.021,Y -472.604,Z 1198.557,A 0.000,B 0.000,C 90.000,E1 100.254} C_DIS
LIN {X 0.065,Y -474.266,Z 1198.556,A 0.000,B 0.000,C 90.000,E1 100.018} C_DIS
LIN {X -0.154,Y -475.651,Z 1198.554,A 0.000,B 0.000,C 90.000,E1 99.792} C_DIS
LIN {X 0.177,Y -476.680,Z 1198.553,A 0.000,B 0.000,C 90.000,E1 99.500} C_DIS
LIN {X -0.086,Y -477.863,Z 1198.550,A 0.000,B 0.000,C 90.000,E1 99.029} C_DIS
LIN {X 0.051,Y -478.042,Z 1198.547,A 0.000,B 0.000,C 90.000,E1 98.511} C_DIS
LIN {X 0.199,Y -477.246,Z 1198.545,A 0.000,B 0.000,C 90.000,E1 97.992} C_DIS
LIN {X -0.123,Y -475.347,Z 1198.542,A 0.000,B 0.000,C 90.000,E1 97.530} C_DIS
LIN {X 0.215,Y -473.870,Z 1198.540,A 0.000,B 0.000,C 90.000,E1 97.239} C_DIS
LIN {X 0.201,Y -455.720,Z 1198.526,A 0.000,B 0.000,C 90.000,E1 94.702} C_DIS
LIN {X -0.148,Y -439.985,Z 1198.513,A 0.000,B 0.000,C 90.000,E1 92.407} C_DIS
LIN {X -0.193,Y -422.389,Z 1198.497,A 0.000,B 0.000,C 90.000,E1 89.484} C_DIS
LIN {X 0.144,Y -412.088,Z 1198.486,A 0.000,B 0.000,C 90.000,E1 87.535} C_DIS
LIN {X -0.077,Y -400.422,Z 1198.474,A 0.000,B 0.000,C 90.000,E1 85.355} C_DIS
LIN {X -0.118,Y -390.226,Z 1198.463,A 0.000,B 0.000,C 90.000,E1 83.394} C_DIS
LIN {X 0.043,Y -381.483,Z 1198.454,A 0.000,B 0.000,C 90.000,E1 81.659} C_DIS
LIN {X 0.034,Y -372.502,Z 1198.444,A 0.000,B 0.000,C 90.000,E1 79.926} C_DIS
LIN {X -0.014,Y -363.194,Z 1198.434,A 0.000,B 0.000,C 90.000,E1 78.173} C_DIS
LIN {X -0.148,Y -353.688,Z 1198.424,A 0.000,B 0.000,C 90.000,E1 76.408} C_DIS
LIN {X -0.106,Y -342.447,Z 1198.413,A 0.000,B 0.000,C 90.000,E1 74.283} C_DIS
LIN {X -0.127,Y -331.247,Z 1198.401,A 0.000,B 0.000,C 90.000,E1 72.127} C_DIS
LIN {X -0.102,Y -314.314,Z 1198.381,A 0.000,B 0.000,C 90.000,E1 68.646} C_DIS
LIN {X -0.013,Y -298.569,Z 1198.361,A 0.000,B 0.000,C 90.000,E1 65.049} C_DIS
LIN {X -0.069,Y -285.324,Z 1198.343,A 0.000,B 0.000,C 90.000,E1 61.719} C_DIS
LIN {X 0.010,Y -272.967,Z 1198.324,A 0.000,B 0.000,C 90.000,E1 58.280} C_DIS
LIN {X 0.052,Y -261.440,Z 1198.304,A 0.000,B 0.000,C 90.000,E1 54.769} C_DIS
LIN {X 0.133,Y -251.671,Z 1198.286,A 0.000,B 0.000,C 90.000,E1 51.537} C_DIS
LIN {X 0.036,Y -241.458,Z 1198.266,A 0.000,B 0.000,C 90.000,E1 47.919} C_DIS
LIN {X 0.010,Y -233.706,Z 1198.250,A 0.000,B 0.000,C 90.000,E1 44.960} C_DIS
LIN {X -0.010,Y -224.537,Z 1198.229,A 0.000,B 0.000,C 90.000,E1 41.191} C_DIS
LIN {X 0.088,Y -217.949,Z 1198.212,A 0.000,B 0.000,C 90.000,E1 38.096} C_DIS
LIN {X 0.088,Y -210.638,Z 1198.190,A 0.000,B 0.000,C 90.000,E1 34.199} C_DIS
LIN {X 0.035,Y -204.207,Z 1198.168,A 0.000,B 0.000,C 90.000,E1 30.256} C_DIS
LIN {X 0.082,Y -198.553,Z 1198.146,A 0.000,B 0.000,C 90.000,E1 26.232} C_DIS
LIN {X -0.033,Y -193.613,Z 1198.123,A 0.000,B 0.000,C 90.000,E1 22.206} C_DIS
LIN {X -0.053,Y -189.525,Z 1198.100,A 0.000,B 0.000,C 90.000,E1 18.109} C_DIS
LIN {X 0.009,Y -185.768,Z 1198.073,A 0.000,B 0.000,C 90.000,E1 13.119} C_DIS
LIN {X -0.065,Y -183.156,Z 1198.040,A 0.000,B 0.000,C 90.000,E1 7.296} C_DIS
LIN {X 0.031,Y -184.292,Z 1197.969,A 0.000,B 0.000,C 90.000,E1 354.489} C_DIS
LIN {X -0.075,Y -187.320,Z 1197.942,A 0.000,B 0.000,C 90.000,E1 349.511} C_DIS
LIN {X 0.007,Y -190.808,Z 1197.919,A 0.000,B 0.000,C 90.000,E1 345.338} C_DIS
LIN {X 0.022,Y -195.293,Z 1197.896,A 0.000,B 0.000,C 90.000,E1 341.221} C_DIS
LIN {X -0.072,Y -200.510,Z 1197.873,A 0.000,B 0.000,C 90.000,E1 337.177} C_DIS
LIN {X 0.024,Y -206.386,Z 1197.851,A 0.000,B 0.000,C 90.000,E1 333.127} C_DIS
LIN {X 0.035,Y -212.792,Z 1197.829,A 0.000,B 0.000,C 90.000,E1 329.154} C_DIS
LIN {X -0.052,Y -219.711,Z 1197.807,A 0.000,B 0.000,C 90.000,E1 325.261} C_DIS
LIN {X 0.058,Y -227.365,Z 1197.786,A 0.000,B 0.000,C 90.000,E1 321.376} C_DIS
LIN {X 0.105,Y -234.212,Z 1197.769,A 0.000,B 0.000,C 90.000,E1 318.324} C_DIS
LIN {X -0.019,Y -241.056,Z 1197.754,A 0.000,B 0.000,C 90.000,E1 315.729} C_DIS
LIN {X 0.020,Y -248.877,Z 1197.740,A 0.000,B 0.000,C 90.000,E1 313.137} C_DIS
LIN {X -0.063,Y -258.947,Z 1197.724,A 0.000,B 0.000,C 90.000,E1 310.253} C_DIS
LIN {X 0.068,Y -271.431,Z 1197.706,A 0.000,B 0.000,C 90.000,E1 307.030} C_DIS
LIN {X 0.061,Y -280.704,Z 1197.694,A 0.000,B 0.000,C 90.000,E1 304.945} C_DIS
LIN {X 0.104,Y -294.300,Z 1197.679,A 0.000,B 0.000,C 90.000,E1 302.212} C_DIS
LIN {X 0.115,Y -303.742,Z 1197.670,A 0.000,B 0.000,C 90.000,E1 300.541} C_DIS
LIN {X -0.094,Y -316.234,Z 1197.659,A 0.000,B 0.000,C 90.000,E1 298.615} C_DIS
LIN {X 0.025,Y -325.312,Z 1197.652,A 0.000,B 0.000,C 90.000,E1 297.308} C_DIS
LIN {X -0.033,Y -335.324,Z 1197.645,A 0.000,B 0.000,C 90.000,E1 296.052} C_DIS
LIN {X 0.008,Y -348.693,Z 1197.636,A 0.000,B 0.000,C 90.000,E1 294.515} C_DIS
LIN {X -0.010,Y -372.438,Z 1197.622,A 0.000,B 0.000,C 90.000,E1 291.972} C_DIS
LIN {X 0.058,Y -391.071,Z 1197.612,A 0.000,B 0.000,C 90.000,E1 290.120} C_DIS
LIN {X 0.106,Y -401.566,Z 1197.606,A 0.000,B 0.000,C 90.000,E1 289.087} C_DIS
LIN {X 0.159,Y -411.924,Z 1197.600,A 0.000,B 0.000,C 90.000,E1 288.055} C_DIS
LIN {X -0.114,Y -422.084,Z 1197.595,A 0.000,B 0.000,C 90.000,E1 287.040} C_DIS
LIN {X -0.055,Y -431.726,Z 1197.589,A 0.000,B 0.000,C 90.000,E1 285.953} C_DIS
LIN {X 0.058,Y -438.381,Z 1197.584,A 0.000,B 0.000,C 90.000,E1 285.134} C_DIS
LIN {X -0.068,Y -444.353,Z 1197.580,A 0.000,B 0.000,C 90.000,E1 284.356} C_DIS
LIN {X 0.175,Y -449.708,Z 1197.575,A 0.000,B 0.000,C 90.000,E1 283.536} C_DIS
LIN {X 0.038,Y -454.389,Z 1197.571,A 0.000,B 0.000,C 90.000,E1 282.771} C_DIS
LIN {X -0.065,Y -458.382,Z 1197.567,A 0.000,B 0.000,C 90.000,E1 282.007} C_DIS
LIN {X 0.038,Y -460.634,Z 1197.564,A 0.000,B 0.000,C 90.000,E1 281.478} C_DIS
LIN {X 0.153,Y -462.594,Z 1197.561,A 0.000,B 0.000,C 90.000,E1 280.950} C_DIS
LIN {X 0.189,Y -464.267,Z 1197.558,A 0.000,B 0.000,C 90.000,E1 280.433} C_DIS
LIN {X -0.136,Y -465.631,Z 1197.555,A 0.000,B 0.000,C 90.000,E1 279.962} C_DIS
LIN {X 0.073,Y -467.653,Z 1197.550,A 0.000,B 0.000,C 90.000,E1 278.916} C_DIS
LIN {X -0.222,Y -469.041,Z 1197.544,A 0.000,B 0.000,C 90.000,E1 277.936} C_DIS
LIN {X -0.069,Y -469.383,Z 1197.541,A 0.000,B 0.000,C 90.000,E1 277.409} C_DIS
LIN {X 0.026,Y -469.361,Z 1197.538,A 0.000,B 0.000,C 90.000,E1 276.891} C_DIS
LIN {X 0.125,Y -468.969,Z 1197.536,A 0.000,B 0.000,C 90.000,E1 276.372} C_DIS
LIN {X 0.221,Y -468.127,Z 1197.533,A 0.000,B 0.000,C 90.000,E1 275.853} C_DIS
LIN {X -0.148,Y -466.782,Z 1197.530,A 0.000,B 0.000,C 90.000,E1 275.391} C_DIS
LIN {X -0.101,Y -465.004,Z 1197.527,A 0.000,B 0.000,C 90.000,E1 274.878} C_DIS
LIN {X -0.018,Y -462.691,Z 1197.524,A 0.000,B 0.000,C 90.000,E1 274.359} C_DIS
LIN {X 0.044,Y -459.724,Z 1197.521,A 0.000,B 0.000,C 90.000,E1 273.841} C_DIS
LIN {X 0.061,Y -455.984,Z 1197.519,A 0.000,B 0.000,C 90.000,E1 273.326} C_DIS
LIN {X -0.141,Y -453.701,Z 1197.517,A 0.000,B 0.000,C 90.000,E1 273.094} C_DIS
LIN {X -0.089,Y -448.307,Z 1197.514,A 0.000,B 0.000,C 90.000,E1 272.579} C_DIS
LIN {X 0.186,Y -445.105,Z 1197.513,A 0.000,B 0.000,C 90.000,E1 272.293} C_DIS
LIN {X -0.140,Y -441.901,Z 1197.512,A 0.000,B 0.000,C 90.000,E1 272.121} C_DIS
LIN {X 0.008,Y -434.916,Z 1197.510,A 0.000,B 0.000,C 90.000,E1 271.718} C_DIS
LIN {X -0.150,Y -427.839,Z 1197.508,A 0.000,B 0.000,C 90.000,E1 271.432} C_DIS
LIN {X 0.085,Y -417.295,Z 1197.506,A 0.000,B 0.000,C 90.000,E1 271.031} C_DIS
LIN {X -0.011,Y -407.452,Z 1197.504,A 0.000,B 0.000,C 90.000,E1 270.745} C_DIS
LIN {X 0.190,Y -396.741,Z 1197.503,A 0.000,B 0.000,C 90.000,E1 270.458} C_DIS
LIN {X 0.011,Y -389.085,Z 1197.502,A 0.000,B 0.000,C 90.000,E1 270.344} C_DIS
LIN {X -0.022,Y -380.380,Z 1197.501,A 0.000,B 0.000,C 90.000,E1 270.229} C_DIS
LIN {X -0.107,Y -372.114,Z 1197.501,A 0.000,B 0.000,C 90.000,E1 270.172} C_DIS
LIN {X 0.111,Y -365.711,Z 1197.501,A 0.000,B 0.000,C 90.000,E1 270.115} C_DIS
LIN {X 0.033,Y -181.575,Z 1197.501,A 0.000,B 0.000,C 90.000,E1 270.115} C_DIS
LIN {X 0.045,Y -180.867,Z 1197.472,A 0.000,B 0.000,C 90.000,E1 265.008} C_DIS
LIN {X -0.078,Y -178.981,Z 1197.444,A 0.000,B 0.000,C 90.000,E1 259.982} C_DIS
LIN {X -0.067,Y -177.953,Z 1197.435,A 0.000,B 0.000,C 90.000,E1 258.285} C_DIS
LIN {X -0.047,Y -175.594,Z 1197.411,A 0.000,B 0.000,C 90.000,E1 254.031} C_DIS
LIN {X -0.034,Y -172.319,Z 1197.387,A 0.000,B 0.000,C 90.000,E1 249.752} C_DIS
LIN {X -0.056,Y -171.797,Z 1197.383,A 0.000,B 0.000,C 90.000,E1 248.901} C_DIS
LIN {X -0.018,Y -169.469,Z 1197.368,A 0.000,B 0.000,C 90.000,E1 246.305} C_DIS
LIN {X 0.038,Y -166.797,Z 1197.349,A 0.000,B 0.000,C 90.000,E1 242.820} C_DIS
LIN {X 0.034,Y -162.777,Z 1197.325,A 0.000,B 0.000,C 90.000,E1 238.456} C_DIS
LIN {X 0.009,Y -161.466,Z 1197.315,A 0.000,B 0.000,C 90.000,E1 236.707} C_DIS
LIN {X 0.049,Y -157.460,Z 1197.291,A 0.000,B 0.000,C 90.000,E1 232.271} C_DIS
LIN {X -0.018,Y -155.472,Z 1197.276,A 0.000,B 0.000,C 90.000,E1 229.622} C_DIS
LIN {X -0.084,Y -151.784,Z 1197.251,A 0.000,B 0.000,C 90.000,E1 225.162} C_DIS
LIN {X -0.071,Y -149.991,Z 1197.236,A 0.000,B 0.000,C 90.000,E1 222.447} C_DIS
LIN {X -0.039,Y -146.823,Z 1197.210,A 0.000,B 0.000,C 90.000,E1 217.890} C_DIS
LIN {X 0.067,Y -145.402,Z 1197.195,A 0.000,B 0.000,C 90.000,E1 215.105} C_DIS
LIN {X -0.016,Y -142.834,Z 1197.170,A 0.000,B 0.000,C 90.000,E1 210.541} C_DIS
LIN {X 0.041,Y -141.448,Z 1197.149,A 0.000,B 0.000,C 90.000,E1 206.821} C_DIS
LIN {X -0.046,Y -139.371,Z 1197.113,A 0.000,B 0.000,C 90.000,E1 200.355} C_DIS
LIN {X 0.071,Y -138.819,Z 1197.097,A 0.000,B 0.000,C 90.000,E1 197.511} C_DIS
LIN {X -0.015,Y -138.353,Z 1197.056,A 0.000,B 0.000,C 90.000,E1 190.074} C_DIS
LIN {X -0.042,Y -139.535,Z 1197.004,A 0.000,B 0.000,C 90.000,E1 180.745} C_DIS
LIN {X 0.051,Y -141.221,Z 1196.973,A 0.000,B 0.000,C 90.000,E1 175.122} C_DIS
LIN {X 0.010,Y -142.594,Z 1196.958,A 0.000,B 0.000,C 90.000,E1 172.356} C_DIS
LIN {X -0.037,Y -144.896,Z 1196.932,A 0.000,B 0.000,C 90.000,E1 167.757} C_DIS
LIN {X -0.083,Y -147.525,Z 1196.911,A 0.000,B 0.000,C 90.000,E1 164.102} C_DIS
LIN {X -0.010,Y -150.121,Z 1196.891,A 0.000,B 0.000,C 90.000,E1 160.423} C_DIS
LIN {X 0.002,Y -153.482,Z 1196.871,A 0.000,B 0.000,C 90.000,E1 156.794} C_DIS
LIN {X 0.065,Y -157.847,Z 1196.846,A 0.000,B 0.000,C 90.000,E1 152.281} C_DIS
LIN {X 0.022,Y -162.131,Z 1196.826,A 0.000,B 0.000,C 90.000,E1 148.742} C_DIS
LIN {X 0.001,Y -166.335,Z 1196.807,A 0.000,B 0.000,C 90.000,E1 145.229} C_DIS
LIN {X 0.008,Y -171.352,Z 1196.787,A 0.000,B 0.000,C 90.000,E1 141.743} C_DIS
LIN {X -0.065,Y -176.257,Z 1196.768,A 0.000,B 0.000,C 90.000,E1 138.324} C_DIS
LIN {X 0.054,Y -180.540,Z 1196.754,A 0.000,B 0.000,C 90.000,E1 135.729} C_DIS
LIN {X 0.033,Y -185.941,Z 1196.735,A 0.000,B 0.000,C 90.000,E1 132.366} C_DIS
LIN {X -0.033,Y -190.572,Z 1196.722,A 0.000,B 0.000,C 90.000,E1 129.886} C_DIS
LIN {X -0.002,Y -196.322,Z 1196.703,A 0.000,B 0.000,C 90.000,E1 126.583} C_DIS
LIN {X 0.068,Y -201.339,Z 1196.689,A 0.000,B 0.000,C 90.000,E1 123.992} C_DIS
LIN {X 0.032,Y -201.574,Z 1196.688,A 0.000,B 0.000,C 90.000,E1 123.865} C_DIS
LIN {X 0.013,Y -311.444,Z 1196.688,A 0.000,B 0.000,C 90.000,E1 123.865} C_DIS
LIN {X -0.037,Y -313.963,Z 1196.688,A 0.000,B 0.000,C 90.000,E1 123.833} C_DIS
LIN {X 0.003,Y -318.801,Z 1196.687,A 0.000,B 0.000,C 90.000,E1 123.579} C_DIS
LIN {X 0.045,Y -321.485,Z 1196.685,A 0.000,B 0.000,C 90.000,E1 123.324} C_DIS
LIN {X -0.132,Y -325.202,Z 1196.682,A 0.000,B 0.000,C 90.000,E1 122.832} C_DIS
LIN {X -0.044,Y -326.774,Z 1196.681,A 0.000,B 0.000,C 90.000,E1 122.498} C_DIS
LIN {X 0.085,Y -340.233,Z 1196.661,A 0.000,B 0.000,C 90.000,E1 119.027} C_DIS
LIN {X -0.015,Y -352.699,Z 1196.646,A 0.000,B 0.000,C 90.000,E1 116.283} C_DIS
LIN {X 0.071,Y -366.671,Z 1196.631,A 0.000,B 0.000,C 90.000,E1 113.567} C_DIS
LIN {X 0.009,Y -380.451,Z 1196.618,A 0.000,B 0.000,C 90.000,E1 111.227} C_DIS
LIN {X 0.167,Y -395.611,Z 1196.605,A 0.000,B 0.000,C 90.000,E1 108.906} C_DIS
LIN {X 0.069,Y -412.259,Z 1196.593,A 0.000,B 0.000,C 90.000,E1 106.677} C_DIS
LIN {X 0.147,Y -430.513,Z 1196.581,A 0.000,B 0.000,C 90.000,E1 104.481} C_DIS
LIN {X -0.083,Y -450.237,Z 1196.569,A 0.000,B 0.000,C 90.000,E1 102.411} C_DIS
LIN {X -0.188,Y -470.592,Z 1196.558,A 0.000,B 0.000,C 90.000,E1 100.489} C_DIS
LIN {X -0.164,Y -472.740,Z 1196.557,A 0.000,B 0.000,C 90.000,E1 100.254} C_DIS
LIN {X -0.141,Y -474.366,Z 1196.556,A 0.000,B 0.000,C 90.000,E1 100.018} C_DIS
LIN {X 0.189,Y -475.704,Z 1196.554,A 0.000,B 0.000,C 90.000,E1 99.726} C_DIS
LIN {X -0.030,Y -476.694,Z 1196.553,A 0.000,B 0.000,C 90.000,E1 99.500} C_DIS
LIN {X 0.179,Y -477.814,Z 1196.550,A 0.000,B 0.000,C 90.000,E1 98.973} C_DIS
LIN {X -0.154,Y -477.935,Z 1196.547,A 0.000,B 0.000,C 90.000,E1 98.511} C_DIS
LIN {X -0.007,Y -477.080,Z 1196.544,A 0.000,B 0.000,C 90.000,E1 97.992} C_DIS
LIN {X 0.143,Y -475.107,Z 1196.542,A 0.000,B 0.000,C 90.000,E1 97.473} C_DIS
LIN {X 0.009,Y -473.580,Z 1196.540,A 0.000,B 0.000,C 90.000,E1 97.239} C_DIS
LIN {X -0.005,Y -455.447,Z 1196.526,A 0.000,B 0.000,C 90.000,E1 94.702} C_DIS
LIN {X -0.098,Y -441.352,Z 1196.515,A 0.000,B 0.000,C 90.000,E1 92.636} C_DIS
LIN {X 0.023,Y -422.094,Z 1196.497,A 0.000,B 0.000,C 90.000,E1 89.427} C_DIS
LIN {X -0.063,Y -411.822,Z 1196.486,A 0.000,B 0.000,C 90.000,E1 87.535} C_DIS
LIN {X 0.113,Y -400.117,Z 1196.474,A 0.000,B 0.000,C 90.000,E1 85.298} C_DIS
LIN {X 0.060,Y -389.927,Z 1196.463,A 0.000,B 0.000,C 90.000,E1 83.337} C_DIS
LIN {X -0.167,Y -381.199,Z 1196.453,A 0.000,B 0.000,C 90.000,E1 81.659} C_DIS
LIN {X -0.111,Y -372.204,Z 1196.444,A 0.000,B 0.000,C 90.000,E1 79.916} C_DIS
LIN {X 0.131,Y -362.884,Z 1196.434,A 0.000,B 0.000,C 90.000,E1 78.117} C_DIS
LIN {X -0.014,Y -353.380,Z 1196.424,A 0.000,B 0.000,C 90.000,E1 76.353} C_DIS
LIN {X 0.107,Y -342.136,Z 1196.412,A 0.000,B 0.000,C 90.000,E1 74.212} C_DIS
LIN {X 0.080,Y -330.932,Z 1196.400,A 0.000,B 0.000,C 90.000,E1 72.054} C_DIS
LIN {X -0.018,Y -314.022,Z 1196.381,A 0.000,B 0.000,C 90.000,E1 68.592} C_DIS
LIN {X 0.175,Y -298.303,Z 1196.361,A 0.000,B 0.000,C 90.000,E1 64.973} C_DIS
LIN {X 0.110,Y -285.056,Z 1196.343,A 0.000,B 0.000,C 90.000,E1 61.641} C_DIS
LIN {X -0.053,Y -272.696,Z 1196.324,A 0.000,B 0.000,C 90.000,E1 58.250} C_DIS
LIN {X -0.003,Y -261.158,Z 1196.304,A 0.000,B 0.000,C 90.000,E1 54.736} C_DIS
LIN {X -0.086,Y -251.328,Z 1196.286,A 0.000,B 0.000,C 90.000,E1 51.537} C_DIS
LIN {X -0.007,Y -241.103,Z 1196.266,A 0.000,B 0.000,C 90.000,E1 47.877} C_DIS
LIN {X -0.048,Y -233.314,Z 1196.250,A 0.000,B 0.000,C 90.000,E1 44.919} C_DIS
LIN {X -0.066,Y -224.194,Z 1196.229,A 0.000,B 0.000,C 90.000,E1 41.148} C_DIS
LIN {X 0.032,Y -217.634,Z 1196.211,A 0.000,B 0.000,C 90.000,E1 38.051} C_DIS
LIN {X 0.000,Y -211.714,Z 1196.194,A 0.000,B 0.000,C 90.000,E1 34.945} C_DIS
LIN {X -0.019,Y -205.128,Z 1196.172,A 0.000,B 0.000,C 90.000,E1 31.003} C_DIS
LIN {X -0.021,Y -199.309,Z 1196.150,A 0.000,B 0.000,C 90.000,E1 27.001} C_DIS
LIN {X -0.030,Y -194.207,Z 1196.127,A 0.000,B 0.000,C 90.000,E1 22.950} C_DIS
LIN {X -0.027,Y -189.926,Z 1196.105,A 0.000,B 0.000,C 90.000,E1 18.852} C_DIS
LIN {X -0.031,Y -186.526,Z 1196.082,A 0.000,B 0.000,C 90.000,E1 14.717} C_DIS
LIN {X -0.065,Y -183.715,Z 1196.054,A 0.000,B 0.000,C 90.000,E1 9.726} C_DIS
LIN {X -0.091,Y -184.345,Z 1195.965,A 0.000,B 0.000,C 90.000,E1 353.685} C_DIS
LIN {X 0.044,Y -187.601,Z 1195.937,A 0.000,B 0.000,C 90.000,E1 348.634} C_DIS
LIN {X -0.053,Y -191.310,Z 1195.914,A 0.000,B 0.000,C 90.000,E1 344.519} C_DIS
LIN {X 0.088,Y -195.961,Z 1195.891,A 0.000,B 0.000,C 90.000,E1 340.369} C_DIS
LIN {X -0.094,Y -201.319,Z 1195.869,A 0.000,B 0.000,C 90.000,E1 336.357} C_DIS
LIN {X 0.026,Y -207.281,Z 1195.846,A 0.000,B 0.000,C 90.000,E1 332.308} C_DIS
LIN {X 0.089,Y -213.807,Z 1195.824,A 0.000,B 0.000,C 90.000,E1 328.329} C_DIS
LIN {X -0.141,Y -220.897,Z 1195.802,A 0.000,B 0.000,C 90.000,E1 324.482} C_DIS
LIN {X 0.002,Y -228.731,Z 1195.781,A 0.000,B 0.000,C 90.000,E1 320.598} C_DIS
LIN {X 0.055,Y -235.869,Z 1195.764,A 0.000,B 0.000,C 90.000,E1 317.553} C_DIS
LIN {X -0.031,Y -243.036,Z 1195.750,A 0.000,B 0.000,C 90.000,E1 314.960} C_DIS
LIN {X 0.068,Y -252.428,Z 1195.733,A 0.000,B 0.000,C 90.000,E1 312.000} C_DIS
LIN {X 0.132,Y -264.327,Z 1195.715,A 0.000,B 0.000,C 90.000,E1 308.749} C_DIS
LIN {X 0.077,Y -274.405,Z 1195.702,A 0.000,B 0.000,C 90.000,E1 306.297} C_DIS
LIN {X -0.087,Y -285.680,Z 1195.688,A 0.000,B 0.000,C 90.000,E1 303.913} C_DIS
LIN {X -0.075,Y -298.060,Z 1195.675,A 0.000,B 0.000,C 90.000,E1 301.544} C_DIS
LIN {X 0.029,Y -309.965,Z 1195.664,A 0.000,B 0.000,C 90.000,E1 299.539} C_DIS
LIN {X 0.136,Y -320.803,Z 1195.655,A 0.000,B 0.000,C 90.000,E1 297.897} C_DIS
LIN {X -0.072,Y -330.239,Z 1195.648,A 0.000,B 0.000,C 90.000,E1 296.668} C_DIS
LIN {X -0.008,Y -340.665,Z 1195.641,A 0.000,B 0.000,C 90.000,E1 295.412} C_DIS
LIN {X 0.000,Y -362.066,Z 1195.628,A 0.000,B 0.000,C 90.000,E1 293.025} C_DIS
LIN {X -0.070,Y -383.661,Z 1195.616,A 0.000,B 0.000,C 90.000,E1 290.844} C_DIS
LIN {X 0.032,Y -396.617,Z 1195.609,A 0.000,B 0.000,C 90.000,E1 289.577} C_DIS
LIN {X -0.141,Y -409.724,Z 1195.602,A 0.000,B 0.000,C 90.000,E1 288.308} C_DIS
LIN {X -0.048,Y -417.437,Z 1195.597,A 0.000,B 0.000,C 90.000,E1 287.511} C_DIS
LIN {X 0.217,Y -424.927,Z 1195.593,A 0.000,B 0.000,C 90.000,E1 286.677} C_DIS
LIN {X -0.020,Y -432.134,Z 1195.588,A 0.000,B 0.000,C 90.000,E1 285.898} C_DIS
LIN {X 0.215,Y -438.763,Z 1195.584,A 0.000,B 0.000,C 90.000,E1 285.064} C_DIS
LIN {X -0.020,Y -444.704,Z 1195.579,A 0.000,B 0.000,C 90.000,E1 284.300} C_DIS
LIN {X -0.209,Y -450.030,Z 1195.575,A 0.000,B 0.000,C 90.000,E1 283.536} C_DIS
LIN {X 0.096,Y -454.680,Z 1195.571,A 0.000,B 0.000,C 90.000,E1 282.715} C_DIS
LIN {X -0.001,Y -458.622,Z 1195.566,A 0.000,B 0.000,C 90.000,E1 281.951} C_DIS
LIN {X 0.103,Y -460.848,Z 1195.563,A 0.000,B 0.000,C 90.000,E1 281.422} C_DIS
LIN {X 0.221,Y -462.780,Z 1195.561,A 0.000,B 0.000,C 90.000,E1 280.894} C_DIS
LIN {X -0.114,Y -464.435,Z 1195.558,A 0.000,B 0.000,C 90.000,E1 280.423} C_DIS
LIN {X -0.063,Y -465.783,Z 1195.555,A 0.000,B 0.000,C 90.000,E1 279.905} C_DIS
LIN {X 0.149,Y -467.790,Z 1195.549,A 0.000,B 0.000,C 90.000,E1 278.859} C_DIS
LIN {X -0.233,Y -468.611,Z 1195.547,A 0.000,B 0.000,C 90.000,E1 278.398} C_DIS
LIN {X -0.080,Y -469.237,Z 1195.544,A 0.000,B 0.000,C 90.000,E1 277.871} C_DIS
LIN {X 0.012,Y -469.583,Z 1195.541,A 0.000,B 0.000,C 90.000,E1 277.352} C_DIS
LIN {X 0.109,Y -469.569,Z 1195.538,A 0.000,B 0.000,C 90.000,E1 276.834} C_DIS
LIN {X 0.208,Y -469.096,Z 1195.535,A 0.000,B 0.000,C 90.000,E1 276.315} C_DIS
LIN {X -0.158,Y -468.222,Z 1195.532,A 0.000,B 0.000,C 90.000,E1 275.853} C_DIS
LIN {X -0.063,Y -466.880,Z 1195.530,A 0.000,B 0.000,C 90.000,E1 275.334} C_DIS
LIN {X -0.013,Y -465.036,Z 1195.527,A 0.000,B 0.000,C 90.000,E1 274.821} C_DIS
LIN {X 0.069,Y -462.654,Z 1195.524,A 0.000,B 0.000,C 90.000,E1 274.302} C_DIS
LIN {X 0.131,Y -459.659,Z 1195.521,A 0.000,B 0.000,C 90.000,E1 273.784} C_DIS
LIN {X 0.147,Y -455.812,Z 1195.518,A 0.000,B 0.000,C 90.000,E1 273.269} C_DIS
LIN {X -0.055,Y -453.547,Z 1195.517,A 0.000,B 0.000,C 90.000,E1 273.037} C_DIS
LIN {X 0.028,Y -448.071,Z 1195.514,A 0.000,B 0.000,C 90.000,E1 272.522} C_DIS
LIN {X -0.110,Y -444.836,Z 1195.513,A 0.000,B 0.000,C 90.000,E1 272.293} C_DIS
LIN {X 0.040,Y -441.735,Z 1195.511,A 0.000,B 0.000,C 90.000,E1 272.064} C_DIS
LIN {X -0.205,Y -434.743,Z 1195.509,A 0.000,B 0.000,C 90.000,E1 271.718} C_DIS
LIN {X 0.081,Y -427.693,Z 1195.508,A 0.000,B 0.000,C 90.000,E1 271.375} C_DIS
LIN {X -0.077,Y -417.235,Z 1195.506,A 0.000,B 0.000,C 90.000,E1 271.031} C_DIS
LIN {X -0.169,Y -407.304,Z 1195.504,A 0.000,B 0.000,C 90.000,E1 270.745} C_DIS
LIN {X 0.035,Y -396.433,Z 1195.503,A 0.000,B 0.000,C 90.000,E1 270.458} C_DIS
LIN {X -0.130,Y -388.792,Z 1195.502,A 0.000,B 0.000,C 90.000,E1 270.344} C_DIS
LIN {X -0.148,Y -380.048,Z 1195.501,A 0.000,B 0.000,C 90.000,E1 270.229} C_DIS
LIN {X 0.076,Y -368.672,Z 1195.501,A 0.000,B 0.000,C 90.000,E1 270.115} C_DIS
LIN {X 0.039,Y -367.239,Z 1195.501,A 0.000,B 0.000,C 90.000,E1 270.115} C_DIS
LIN {X 0.001,Y -181.574,Z 1195.501,A 0.000,B 0.000,C 90.000,E1 270.115} C_DIS
LIN {X -0.063,Y -180.908,Z 1195.475,A 0.000,B 0.000,C 90.000,E1 265.584} C_DIS
LIN {X -0.006,Y -180.776,Z 1195.471,A 0.000,B 0.000,C 90.000,E1 264.723} C_DIS
LIN {X 0.065,Y -178.872,Z 1195.443,A 0.000,B 0.000,C 90.000,E1 259.634} C_DIS
LIN {X -0.034,Y -175.914,Z 1195.414,A 0.000,B 0.000,C 90.000,E1 254.574} C_DIS
LIN {X 0.022,Y -174.605,Z 1195.405,A 0.000,B 0.000,C 90.000,E1 252.851} C_DIS
LIN {X -0.052,Y -171.587,Z 1195.381,A 0.000,B 0.000,C 90.000,E1 248.592} C_DIS
LIN {X -0.062,Y -167.810,Z 1195.357,A 0.000,B 0.000,C 90.000,E1 244.280} C_DIS
LIN {X -0.045,Y -166.530,Z 1195.347,A 0.000,B 0.000,C 90.000,E1 242.538} C_DIS
LIN {X 0.091,Y -162.529,Z 1195.323,A 0.000,B 0.000,C 90.000,E1 238.122} C_DIS
LIN {X -0.073,Y -161.204,Z 1195.313,A 0.000,B 0.000,C 90.000,E1 236.421} C_DIS
LIN {X -0.037,Y -157.214,Z 1195.289,A 0.000,B 0.000,C 90.000,E1 231.984} C_DIS
LIN {X -0.014,Y -155.940,Z 1195.279,A 0.000,B 0.000,C 90.000,E1 230.194} C_DIS
LIN {X -0.053,Y -152.192,Z 1195.254,A 0.000,B 0.000,C 90.000,E1 225.729} C_DIS
LIN {X -0.032,Y -150.439,Z 1195.239,A 0.000,B 0.000,C 90.000,E1 223.014} C_DIS
LIN {X -0.005,Y -147.165,Z 1195.214,A 0.000,B 0.000,C 90.000,E1 218.463} C_DIS
LIN {X -0.038,Y -145.182,Z 1195.193,A 0.000,B 0.000,C 90.000,E1 214.818} C_DIS
LIN {X -0.003,Y -142.326,Z 1195.163,A 0.000,B 0.000,C 90.000,E1 209.283} C_DIS
LIN {X -0.008,Y -141.716,Z 1195.152,A 0.000,B 0.000,C 90.000,E1 207.436} C_DIS
LIN {X 0.039,Y -139.475,Z 1195.116,A 0.000,B 0.000,C 90.000,E1 200.918} C_DIS
LIN {X 0.031,Y -138.971,Z 1195.101,A 0.000,B 0.000,C 90.000,E1 198.127} C_DIS
LIN {X 0.019,Y -138.330,Z 1195.054,A 0.000,B 0.000,C 90.000,E1 189.726} C_DIS
LIN {X 0.023,Y -139.436,Z 1195.007,A 0.000,B 0.000,C 90.000,E1 181.318} C_DIS
LIN {X -0.038,Y -140.967,Z 1194.976,A 0.000,B 0.000,C 90.000,E1 175.755} C_DIS
LIN {X 0.054,Y -142.722,Z 1194.956,A 0.000,B 0.000,C 90.000,E1 172.008} C_DIS
LIN {X 0.011,Y -145.104,Z 1194.930,A 0.000,B 0.000,C 90.000,E1 167.409} C_DIS
LIN {X 0.006,Y -147.728,Z 1194.910,A 0.000,B 0.000,C 90.000,E1 163.740} C_DIS
LIN {X -0.053,Y -150.389,Z 1194.889,A 0.000,B 0.000,C 90.000,E1 160.115} C_DIS
LIN {X -0.036,Y -153.822,Z 1194.869,A 0.000,B 0.000,C 90.000,E1 156.485} C_DIS
LIN {X 0.023,Y -157.234,Z 1194.849,A 0.000,B 0.000,C 90.000,E1 152.871} C_DIS
LIN {X -0.037,Y -161.402,Z 1194.830,A 0.000,B 0.000,C 90.000,E1 149.331} C_DIS
LIN {X -0.027,Y -165.604,Z 1194.810,A 0.000,B 0.000,C 90.000,E1 145.801} C_DIS
LIN {X -0.041,Y -170.529,Z 1194.791,A 0.000,B 0.000,C 90.000,E1 142.316} C_DIS
LIN {X 0.003,Y -175.408,Z 1194.771,A 0.000,B 0.000,C 90.000,E1 138.852} C_DIS
LIN {X -0.006,Y -181.033,Z 1194.752,A 0.000,B 0.000,C 90.000,E1 135.445} C_DIS
LIN {X -0.013,Y -186.466,Z 1194.734,A 0.000,B 0.000,C 90.000,E1 132.081} C_DIS
LIN {X 0.056,Y -191.089,Z 1194.720,A 0.000,B 0.000,C 90.000,E1 129.564} C_DIS
LIN {X -0.023,Y -196.879,Z 1194.702,A 0.000,B 0.000,C 90.000,E1 126.297} C_DIS
LIN {X -0.052,Y -201.181,Z 1194.689,A 0.000,B 0.000,C 90.000,E1 124.119} C_DIS
LIN {X -0.080,Y -201.547,Z 1194.688,A 0.000,B 0.000,C 90.000,E1 123.913} C_DIS
LIN {X 0.083,Y -312.249,Z 1194.688,A 0.000,B 0.000,C 90.000,E1 123.865} C_DIS
LIN {X -0.076,Y -313.717,Z 1194.688,A 0.000,B 0.000,C 90.000,E1 123.865} C_DIS
LIN {X -0.017,Y -317.180,Z 1194.687,A 0.000,B 0.000,C 90.000,E1 123.706} C_DIS
LIN {X -0.084,Y -320.580,Z 1194.686,A 0.000,B 0.000,C 90.000,E1 123.452} C_DIS
LIN {X 0.101,Y -324.227,Z 1194.683,A 0.000,B 0.000,C 90.000,E1 122.959} C_DIS
LIN {X -0.087,Y -325.998,Z 1194.681,A 0.000,B 0.000,C 90.000,E1 122.673} C_DIS
LIN {X 0.101,Y -328.525,Z 1194.678,A 0.000,B 0.000,C 90.000,E1 122.005} C_DIS
LIN {X 0.000,Y -339.523,Z 1194.662,A 0.000,B 0.000,C 90.000,E1 119.205} C_DIS
LIN {X 0.027,Y -351.904,Z 1194.647,A 0.000,B 0.000,C 90.000,E1 116.437} C_DIS
LIN {X -0.228,Y -365.786,Z 1194.632,A 0.000,B 0.000,C 90.000,E1 113.770} C_DIS
LIN {X -0.173,Y -379.477,Z 1194.619,A 0.000,B 0.000,C 90.000,E1 111.408} C_DIS
LIN {X -0.049,Y -394.543,Z 1194.606,A 0.000,B 0.000,C 90.000,E1 109.087} C_DIS
LIN {X -0.183,Y -411.089,Z 1194.594,A 0.000,B 0.000,C 90.000,E1 106.858} C_DIS
LIN {X -0.035,Y -429.233,Z 1194.581,A 0.000,B 0.000,C 90.000,E1 104.647} C_DIS
LIN {X -0.016,Y -448.892,Z 1194.570,A 0.000,B 0.000,C 90.000,E1 102.535} C_DIS
LIN {X -0.070,Y -471.635,Z 1194.557,A 0.000,B 0.000,C 90.000,E1 100.366} C_DIS
LIN {X -0.110,Y -473.486,Z 1194.556,A 0.000,B 0.000,C 90.000,E1 100.141} C_DIS
LIN {X 0.217,Y -475.025,Z 1194.555,A 0.000,B 0.000,C 90.000,E1 99.849} C_DIS
LIN {X 0.076,Y -476.175,Z 1194.553,A 0.000,B 0.000,C 90.000,E1 99.613} C_DIS
LIN {X 0.205,Y -477.556,Z 1194.551,A 0.000,B 0.000,C 90.000,E1 99.095} C_DIS
LIN {X -0.058,Y -477.910,Z 1194.548,A 0.000,B 0.000,C 90.000,E1 98.624} C_DIS
LIN {X 0.087,Y -477.295,Z 1194.545,A 0.000,B 0.000,C 90.000,E1 98.106} C_DIS
LIN {X -0.237,Y -475.616,Z 1194.542,A 0.000,B 0.000,C 90.000,E1 97.644} C_DIS
LIN {X 0.102,Y -474.285,Z 1194.541,A 0.000,B 0.000,C 90.000,E1 97.352} C_DIS
LIN {X 0.051,Y -459.779,Z 1194.530,A 0.000,B 0.000,C 90.000,E1 95.334} C_DIS
LIN {X -0.167,Y -443.762,Z 1194.517,A 0.000,B 0.000,C 90.000,E1 93.037} C_DIS
LIN {X 0.033,Y -424.229,Z 1194.499,A 0.000,B 0.000,C 90.000,E1 89.828} C_DIS
LIN {X 0.080,Y -412.415,Z 1194.487,A 0.000,B 0.000,C 90.000,E1 87.650} C_DIS
LIN {X -0.184,Y -402.155,Z 1194.476,A 0.000,B 0.000,C 90.000,E1 85.755} C_DIS
LIN {X 0.172,Y -391.962,Z 1194.465,A 0.000,B 0.000,C 90.000,E1 83.742} C_DIS
LIN {X -0.047,Y -381.788,Z 1194.454,A 0.000,B 0.000,C 90.000,E1 81.781} C_DIS
LIN {X 0.008,Y -372.811,Z 1194.445,A 0.000,B 0.000,C 90.000,E1 80.038} C_DIS
LIN {X -0.009,Y -365.098,Z 1194.437,A 0.000,B 0.000,C 90.000,E1 78.578} C_DIS
LIN {X 0.193,Y -354.009,Z 1194.425,A 0.000,B 0.000,C 90.000,E1 76.464} C_DIS
LIN {X -0.096,Y -342.779,Z 1194.413,A 0.000,B 0.000,C 90.000,E1 74.393} C_DIS
LIN {X -0.104,Y -331.562,Z 1194.401,A 0.000,B 0.000,C 90.000,E1 72.236} C_DIS
LIN {X 0.122,Y -314.609,Z 1194.382,A 0.000,B 0.000,C 90.000,E1 68.720} C_DIS
LIN {X -0.071,Y -298.838,Z 1194.362,A 0.000,B 0.000,C 90.000,E1 65.177} C_DIS
LIN {X 0.017,Y -285.563,Z 1194.344,A 0.000,B 0.000,C 90.000,E1 61.820} C_DIS
LIN {X -0.027,Y -273.138,Z 1194.324,A 0.000,B 0.000,C 90.000,E1 58.408} C_DIS
LIN {X 0.026,Y -261.536,Z 1194.305,A 0.000,B 0.000,C 90.000,E1 54.895} C_DIS
LIN {X -0.062,Y -251.627,Z 1194.287,A 0.000,B 0.000,C 90.000,E1 51.698} C_DIS
LIN {X 0.022,Y -241.341,Z 1194.267,A 0.000,B 0.000,C 90.000,E1 48.038} C_DIS
LIN {X -0.094,Y -231.632,Z 1194.246,A 0.000,B 0.000,C 90.000,E1 44.352} C_DIS
LIN {X 0.001,Y -222.685,Z 1194.225,A 0.000,B 0.000,C 90.000,E1 40.539} C_DIS
LIN {X 0.056,Y -216.269,Z 1194.208,A 0.000,B 0.000,C 90.000,E1 37.443} C_DIS
LIN {X 0.032,Y -210.455,Z 1194.191,A 0.000,B 0.000,C 90.000,E1 34.326} C_DIS
LIN {X -0.027,Y -203.980,Z 1194.169,A 0.000,B 0.000,C 90.000,E1 30.384} C_DIS
LIN {X 0.012,Y -198.217,Z 1194.146,A 0.000,B 0.000,C 90.000,E1 26.360} C_DIS
LIN {X 0.069,Y -193.222,Z 1194.124,A 0.000,B 0.000,C 90.000,E1 22.280} C_DIS
LIN {X 0.043,Y -189.021,Z 1194.101,A 0.000,B 0.000,C 90.000,E1 18.181} C_DIS
LIN {X -0.042,Y -185.217,Z 1194.073,A 0.000,B 0.000,C 90.000,E1 13.231} C_DIS
LIN {X 0.035,Y -182.554,Z 1194.041,A 0.000,B 0.000,C 90.000,E1 7.352} C_DIS
LIN {X 0.005,Y -183.583,Z 1193.969,A 0.000,B 0.000,C 90.000,E1 354.489} C_DIS
LIN {X 0.057,Y -186.617,Z 1193.942,A 0.000,B 0.000,C 90.000,E1 349.454} C_DIS
LIN {X -0.068,Y -190.146,Z 1193.918,A 0.000,B 0.000,C 90.000,E1 345.338} C_DIS
LIN {X -0.075,Y -194.632,Z 1193.896,A 0.000,B 0.000,C 90.000,E1 341.221} C_DIS
LIN {X 0.070,Y -199.876,Z 1193.873,A 0.000,B 0.000,C 90.000,E1 337.102} C_DIS
LIN {X 0.063,Y -205.728,Z 1193.850,A 0.000,B 0.000,C 90.000,E1 333.076} C_DIS
LIN {X -0.027,Y -212.128,Z 1193.828,A 0.000,B 0.000,C 90.000,E1 329.125} C_DIS
LIN {X 0.058,Y -219.116,Z 1193.807,A 0.000,B 0.000,C 90.000,E1 325.182} C_DIS
LIN {X 0.013,Y -226.809,Z 1193.785,A 0.000,B 0.000,C 90.000,E1 321.331} C_DIS
LIN {X -0.137,Y -233.764,Z 1193.768,A 0.000,B 0.000,C 90.000,E1 318.324} C_DIS
LIN {X 0.063,Y -240.719,Z 1193.754,A 0.000,B 0.000,C 90.000,E1 315.648} C_DIS
LIN {X -0.074,Y -248.696,Z 1193.739,A 0.000,B 0.000,C 90.000,E1 313.095} C_DIS
LIN {X 0.051,Y -260.172,Z 1193.721,A 0.000,B 0.000,C 90.000,E1 309.806} C_DIS
LIN {X -0.002,Y -272.877,Z 1193.703,A 0.000,B 0.000,C 90.000,E1 306.629} C_DIS
LIN {X 0.078,Y -282.357,Z 1193.692,A 0.000,B 0.000,C 90.000,E1 304.532} C_DIS
LIN {X 0.166,Y -296.305,Z 1193.677,A 0.000,B 0.000,C 90.000,E1 301.799} C_DIS
LIN {X -0.180,Y -308.026,Z 1193.666,A 0.000,B 0.000,C 90.000,E1 299.873} C_DIS
LIN {X -0.104,Y -318.681,Z 1193.657,A 0.000,B 0.000,C 90.000,E1 298.231} C_DIS
LIN {X 0.063,Y -327.920,Z 1193.650,A 0.000,B 0.000,C 90.000,E1 296.924} C_DIS
LIN {X 0.073,Y -338.125,Z 1193.643,A 0.000,B 0.000,C 90.000,E1 295.668} C_DIS
LIN {X 0.057,Y -356.715,Z 1193.631,A 0.000,B 0.000,C 90.000,E1 293.567} C_DIS
LIN {X -0.034,Y -380.815,Z 1193.617,A 0.000,B 0.000,C 90.000,E1 291.099} C_DIS
LIN {X -0.201,Y -396.869,Z 1193.609,A 0.000,B 0.000,C 90.000,E1 289.577} C_DIS
LIN {X 0.145,Y -409.997,Z 1193.601,A 0.000,B 0.000,C 90.000,E1 288.236} C_DIS
LIN {X -0.082,Y -420.193,Z 1193.596,A 0.000,B 0.000,C 90.000,E1 287.221} C_DIS
LIN {X -0.189,Y -427.506,Z 1193.591,A 0.000,B 0.000,C 90.000,E1 286.441} C_DIS
LIN {X 0.099,Y -434.419,Z 1193.587,A 0.000,B 0.000,C 90.000,E1 285.607} C_DIS
LIN {X -0.060,Y -440.864,Z 1193.582,A 0.000,B 0.000,C 90.000,E1 284.828} C_DIS
LIN {X 0.147,Y -446.632,Z 1193.578,A 0.000,B 0.000,C 90.000,E1 284.008} C_DIS
LIN {X -0.016,Y -451.709,Z 1193.574,A 0.000,B 0.000,C 90.000,E1 283.244} C_DIS
LIN {X -0.141,Y -456.162,Z 1193.569,A 0.000,B 0.000,C 90.000,E1 282.479} C_DIS
LIN {X -0.225,Y -459.832,Z 1193.565,A 0.000,B 0.000,C 90.000,E1 281.715} C_DIS
LIN {X 0.170,Y -462.854,Z 1193.561,A 0.000,B 0.000,C 90.000,E1 280.894} C_DIS
LIN {X -0.163,Y -464.500,Z 1193.558,A 0.000,B 0.000,C 90.000,E1 280.423} C_DIS
LIN {X -0.114,Y -465.843,Z 1193.555,A 0.000,B 0.000,C 90.000,E1 279.905} C_DIS
LIN {X 0.099,Y -467.920,Z 1193.549,A 0.000,B 0.000,C 90.000,E1 278.859} C_DIS
LIN {X 0.181,Y -468.783,Z 1193.547,A 0.000,B 0.000,C 90.000,E1 278.341} C_DIS
LIN {X -0.128,Y -469.440,Z 1193.544,A 0.000,B 0.000,C 90.000,E1 277.871} C_DIS
LIN {X -0.035,Y -469.813,Z 1193.541,A 0.000,B 0.000,C 90.000,E1 277.352} C_DIS
LIN {X 0.062,Y -469.798,Z 1193.538,A 0.000,B 0.000,C 90.000,E1 276.834} C_DIS
LIN {X 0.163,Y -469.347,Z 1193.535,A 0.000,B 0.000,C 90.000,E1 276.315} C_DIS
LIN {X -0.202,Y -468.473,Z 1193.532,A 0.000,B 0.000,C 90.000,E1 275.853} C_DIS
LIN {X -0.105,Y -467.094,Z 1193.530,A 0.000,B 0.000,C 90.000,E1 275.334} C_DIS
LIN {X -0.054,Y -465.245,Z 1193.527,A 0.000,B 0.000,C 90.000,E1 274.821} C_DIS
LIN {X 0.030,Y -462.858,Z 1193.524,A 0.000,B 0.000,C 90.000,E1 274.302} C_DIS
LIN {X 0.093,Y -459.829,Z 1193.521,A 0.000,B 0.000,C 90.000,E1 273.784} C_DIS
LIN {X 0.111,Y -456.006,Z 1193.518,A 0.000,B 0.000,C 90.000,E1 273.269} C_DIS
LIN {X -0.091,Y -453.739,Z 1193.517,A 0.000,B 0.000,C 90.000,E1 273.037} C_DIS
LIN {X 0.135,Y -451.123,Z 1193.515,A 0.000,B 0.000,C 90.000,E1 272.751} C_DIS
LIN {X -0.020,Y -448.274,Z 1193.514,A 0.000,B 0.000,C 90.000,E1 272.522} C_DIS
LIN {X -0.171,Y -445.031,Z 1193.513,A 0.000,B 0.000,C 90.000,E1 272.293} C_DIS
LIN {X -0.027,Y -441.925,Z 1193.511,A 0.000,B 0.000,C 90.000,E1 272.064} C_DIS
LIN {X 0.117,Y -438.323,Z 1193.510,A 0.000,B 0.000,C 90.000,E1 271.835} C_DIS
LIN {X 0.146,Y -431.198,Z 1193.508,A 0.000,B 0.000,C 90.000,E1 271.489} C_DIS
LIN {X -0.184,Y -420.924,Z 1193.506,A 0.000,B 0.000,C 90.000,E1 271.146} C_DIS
LIN {X 0.012,Y -410.899,Z 1193.505,A 0.000,B 0.000,C 90.000,E1 270.802} C_DIS
LIN {X 0.120,Y -400.375,Z 1193.503,A 0.000,B 0.000,C 90.000,E1 270.516} C_DIS
LIN {X 0.179,Y -389.041,Z 1193.502,A 0.000,B 0.000,C 90.000,E1 270.286} C_DIS
LIN {X 0.164,Y -380.495,Z 1193.501,A 0.000,B 0.000,C 90.000,E1 270.172} C_DIS
LIN {X 0.008,Y -369.460,Z 1193.501,A 0.000,B 0.000,C 90.000,E1 270.115} C_DIS
LIN {X -0.066,Y -364.666,Z 1193.501,A 0.000,B 0.000,C 90.000,E1 270.115} C_DIS
LIN {X -0.053,Y -181.573,Z 1193.500,A 0.000,B 0.000,C 90.000,E1 270.115} C_DIS
LIN {X -0.027,Y -180.861,Z 1193.472,A 0.000,B 0.000,C 90.000,E1 265.008} C_DIS
LIN {X 0.027,Y -178.975,Z 1193.444,A 0.000,B 0.000,C 90.000,E1 259.926} C_DIS
LIN {X 0.037,Y -177.937,Z 1193.435,A 0.000,B 0.000,C 90.000,E1 258.229} C_DIS
LIN {X 0.051,Y -175.577,Z 1193.411,A 0.000,B 0.000,C 90.000,E1 253.976} C_DIS
LIN {X 0.058,Y -172.304,Z 1193.387,A 0.000,B 0.000,C 90.000,E1 249.699} C_DIS
LIN {X 0.035,Y -171.783,Z 1193.383,A 0.000,B 0.000,C 90.000,E1 248.847} C_DIS
LIN {X -0.019,Y -169.448,Z 1193.368,A 0.000,B 0.000,C 90.000,E1 246.282} C_DIS
LIN {X 0.045,Y -166.778,Z 1193.349,A 0.000,B 0.000,C 90.000,E1 242.794} C_DIS
LIN {X -0.035,Y -162.758,Z 1193.325,A 0.000,B 0.000,C 90.000,E1 238.456} C_DIS
LIN {X -0.059,Y -161.448,Z 1193.315,A 0.000,B 0.000,C 90.000,E1 236.707} C_DIS
LIN {X -0.016,Y -157.441,Z 1193.290,A 0.000,B 0.000,C 90.000,E1 232.271} C_DIS
LIN {X 0.017,Y -155.449,Z 1193.276,A 0.000,B 0.000,C 90.000,E1 229.585} C_DIS
LIN {X 0.066,Y -151.767,Z 1193.251,A 0.000,B 0.000,C 90.000,E1 225.081} C_DIS
LIN {X 0.077,Y -149.970,Z 1193.235,A 0.000,B 0.000,C 90.000,E1 222.366} C_DIS
LIN {X -0.012,Y -146.808,Z 1193.210,A 0.000,B 0.000,C 90.000,E1 217.855} C_DIS
LIN {X 0.004,Y -145.385,Z 1193.195,A 0.000,B 0.000,C 90.000,E1 215.105} C_DIS
LIN {X -0.005,Y -142.443,Z 1193.164,A 0.000,B 0.000,C 90.000,E1 209.589} C_DIS
LIN {X -0.021,Y -141.435,Z 1193.149,A 0.000,B 0.000,C 90.000,E1 206.821} C_DIS
LIN {X 0.023,Y -139.366,Z 1193.113,A 0.000,B 0.000,C 90.000,E1 200.301} C_DIS
LIN {X 0.010,Y -138.813,Z 1193.097,A 0.000,B 0.000,C 90.000,E1 197.511} C_DIS
LIN {X 0.060,Y -138.351,Z 1193.056,A 0.000,B 0.000,C 90.000,E1 190.018} C_DIS
LIN {X 0.036,Y -139.538,Z 1193.004,A 0.000,B 0.000,C 90.000,E1 180.688} C_DIS
LIN {X -0.011,Y -141.232,Z 1192.973,A 0.000,B 0.000,C 90.000,E1 175.122} C_DIS
LIN {X -0.053,Y -142.603,Z 1192.957,A 0.000,B 0.000,C 90.000,E1 172.356} C_DIS
LIN {X 0.042,Y -144.912,Z 1192.932,A 0.000,B 0.000,C 90.000,E1 167.701} C_DIS
LIN {X 0.035,Y -147.540,Z 1192.911,A 0.000,B 0.000,C 90.000,E1 164.031} C_DIS
LIN {X 0.068,Y -150.141,Z 1192.891,A 0.000,B 0.000,C 90.000,E1 160.369} C_DIS
LIN {X -0.064,Y -153.508,Z 1192.871,A 0.000,B 0.000,C 90.000,E1 156.794} C_DIS
LIN {X -0.001,Y -157.872,Z 1192.846,A 0.000,B 0.000,C 90.000,E1 152.281} C_DIS
LIN {X -0.046,Y -162.160,Z 1192.826,A 0.000,B 0.000,C 90.000,E1 148.742} C_DIS
LIN {X 0.069,Y -166.367,Z 1192.807,A 0.000,B 0.000,C 90.000,E1 145.182} C_DIS
LIN {X -0.063,Y -171.383,Z 1192.787,A 0.000,B 0.000,C 90.000,E1 141.743} C_DIS
LIN {X 0.113,Y -176.293,Z 1192.768,A 0.000,B 0.000,C 90.000,E1 138.243} C_DIS
LIN {X -0.019,Y -180.580,Z 1192.754,A 0.000,B 0.000,C 90.000,E1 135.729} C_DIS
LIN {X -0.041,Y -185.981,Z 1192.735,A 0.000,B 0.000,C 90.000,E1 132.366} C_DIS
LIN {X 0.015,Y -190.614,Z 1192.721,A 0.000,B 0.000,C 90.000,E1 129.850} C_DIS
LIN {X -0.078,Y -196.364,Z 1192.703,A 0.000,B 0.000,C 90.000,E1 126.583} C_DIS
LIN {X -0.009,Y -201.376,Z 1192.689,A 0.000,B 0.000,C 90.000,E1 123.992} C_DIS
LIN {X 0.028,Y -201.495,Z 1192.688,A 0.000,B 0.000,C 90.000,E1 123.913} C_DIS
LIN {X 0.008,Y -311.585,Z 1192.688,A 0.000,B 0.000,C 90.000,E1 123.913} C_DIS
LIN {X 0.002,Y -314.057,Z 1192.688,A 0.000,B 0.000,C 90.000,E1 123.865} C_DIS
LIN {X 0.051,Y -319.067,Z 1192.687,A 0.000,B 0.000,C 90.000,E1 123.579} C_DIS
LIN {X 0.098,Y -321.864,Z 1192.685,A 0.000,B 0.000,C 90.000,E1 123.293} C_DIS
LIN {X 0.016,Y -325.519,Z 1192.682,A 0.000,B 0.000,C 90.000,E1 122.752} C_DIS
LIN {X 0.106,Y -326.976,Z 1192.680,A 0.000,B 0.000,C 90.000,E1 122.418} C_DIS
LIN {X 0.099,Y -339.106,Z 1192.663,A 0.000,B 0.000,C 90.000,E1 119.283} C_DIS
LIN {X -0.038,Y -351.442,Z 1192.647,A 0.000,B 0.000,C 90.000,E1 116.539} C_DIS
LIN {X 0.016,Y -365.266,Z 1192.632,A 0.000,B 0.000,C 90.000,E1 113.823} C_DIS
LIN {X 0.061,Y -378.906,Z 1192.619,A 0.000,B 0.000,C 90.000,E1 111.461} C_DIS
LIN {X 0.174,Y -393.918,Z 1192.606,A 0.000,B 0.000,C 90.000,E1 109.141} C_DIS
LIN {X 0.030,Y -410.405,Z 1192.594,A 0.000,B 0.000,C 90.000,E1 106.913} C_DIS
LIN {X 0.056,Y -428.485,Z 1192.582,A 0.000,B 0.000,C 90.000,E1 104.717} C_DIS
LIN {X 0.161,Y -448.089,Z 1192.570,A 0.000,B 0.000,C 90.000,E1 102.591} C_DIS
LIN {X -0.052,Y -470.937,Z 1192.558,A 0.000,B 0.000,C 90.000,E1 100.433} C_DIS
LIN {X -0.043,Y -472.969,Z 1192.557,A 0.000,B 0.000,C 90.000,E1 100.197} C_DIS
LIN {X -0.035,Y -474.514,Z 1192.555,A 0.000,B 0.000,C 90.000,E1 99.962} C_DIS
LIN {X -0.173,Y -475.773,Z 1192.554,A 0.000,B 0.000,C 90.000,E1 99.726} C_DIS
LIN {X 0.079,Y -476.697,Z 1192.552,A 0.000,B 0.000,C 90.000,E1 99.443} C_DIS
LIN {X -0.183,Y -477.706,Z 1192.550,A 0.000,B 0.000,C 90.000,E1 98.973} C_DIS
LIN {X -0.044,Y -477.728,Z 1192.547,A 0.000,B 0.000,C 90.000,E1 98.454} C_DIS
LIN {X 0.103,Y -476.766,Z 1192.544,A 0.000,B 0.000,C 90.000,E1 97.936} C_DIS
LIN {X -0.157,Y -474.660,Z 1192.541,A 0.000,B 0.000,C 90.000,E1 97.466} C_DIS
LIN {X 0.118,Y -473.039,Z 1192.540,A 0.000,B 0.000,C 90.000,E1 97.182} C_DIS
LIN {X -0.176,Y -456.685,Z 1192.527,A 0.000,B 0.000,C 90.000,E1 94.935} C_DIS
LIN {X -0.021,Y -440.818,Z 1192.514,A 0.000,B 0.000,C 90.000,E1 92.579} C_DIS
LIN {X -0.042,Y -423.080,Z 1192.498,A 0.000,B 0.000,C 90.000,E1 89.656} C_DIS
LIN {X -0.110,Y -412.773,Z 1192.488,A 0.000,B 0.000,C 90.000,E1 87.764} C_DIS
LIN {X 0.045,Y -402.504,Z 1192.477,A 0.000,B 0.000,C 90.000,E1 85.812} C_DIS
LIN {X 0.025,Y -390.848,Z 1192.464,A 0.000,B 0.000,C 90.000,E1 83.571} C_DIS
LIN {X -0.161,Y -380.652,Z 1192.453,A 0.000,B 0.000,C 90.000,E1 81.602} C_DIS
LIN {X -0.118,Y -371.636,Z 1192.444,A 0.000,B 0.000,C 90.000,E1 79.859} C_DIS
LIN {X 0.211,Y -363.895,Z 1192.435,A 0.000,B 0.000,C 90.000,E1 78.342} C_DIS
LIN {X 0.008,Y -354.373,Z 1192.426,A 0.000,B 0.000,C 90.000,E1 76.589} C_DIS
LIN {X 0.053,Y -343.133,Z 1192.414,A 0.000,B 0.000,C 90.000,E1 74.464} C_DIS
LIN {X 0.044,Y -331.923,Z 1192.402,A 0.000,B 0.000,C 90.000,E1 72.308} C_DIS
LIN {X 0.031,Y -316.445,Z 1192.384,A 0.000,B 0.000,C 90.000,E1 69.156} C_DIS
LIN {X -0.099,Y -300.511,Z 1192.364,A 0.000,B 0.000,C 90.000,E1 65.613} C_DIS
LIN {X -0.089,Y -287.126,Z 1192.346,A 0.000,B 0.000,C 90.000,E1 62.281} C_DIS
LIN {X -0.081,Y -274.589,Z 1192.327,A 0.000,B 0.000,C 90.000,E1 58.869} C_DIS
LIN {X -0.125,Y -262.844,Z 1192.308,A 0.000,B 0.000,C 90.000,E1 55.388} C_DIS
LIN {X 0.152,Y -253.926,Z 1192.292,A 0.000,B 0.000,C 90.000,E1 52.477} C_DIS
LIN {X -0.020,Y -244.440,Z 1192.274,A 0.000,B 0.000,C 90.000,E1 49.256} C_DIS
LIN {X 0.028,Y -236.460,Z 1192.257,A 0.000,B 0.000,C 90.000,E1 46.296} C_DIS
LIN {X 0.092,Y -227.105,Z 1192.236,A 0.000,B 0.000,C 90.000,E1 42.528} C_DIS
LIN {X 0.056,Y -220.246,Z 1192.219,A 0.000,B 0.000,C 90.000,E1 39.483} C_DIS
LIN {X 0.081,Y -212.568,Z 1192.198,A 0.000,B 0.000,C 90.000,E1 35.598} C_DIS
LIN {X 0.028,Y -205.829,Z 1192.176,A 0.000,B 0.000,C 90.000,E1 31.671} C_DIS
LIN {X -0.034,Y -199.797,Z 1192.154,A 0.000,B 0.000,C 90.000,E1 27.692} C_DIS
LIN {X -0.033,Y -194.505,Z 1192.131,A 0.000,B 0.000,C 90.000,E1 23.643} C_DIS
LIN {X 0.048,Y -190.016,Z 1192.109,A 0.000,B 0.000,C 90.000,E1 19.523} C_DIS
LIN {X -0.078,Y -186.398,Z 1192.086,A 0.000,B 0.000,C 90.000,E1 15.426} C_DIS
LIN {X 0.101,Y -183.392,Z 1192.058,A 0.000,B 0.000,C 90.000,E1 10.366} C_DIS
LIN {X 0.033,Y -181.560,Z 1192.006,A 0.000,B 0.000,C 90.000,E1 1.146} C_DIS
LIN {X 0.062,Y -183.632,Z 1191.965,A 0.000,B 0.000,C 90.000,E1 353.628} C_DIS
LIN {X -0.012,Y -186.890,Z 1191.937,A 0.000,B 0.000,C 90.000,E1 348.634} C_DIS
LIN {X 0.051,Y -190.642,Z 1191.914,A 0.000,B 0.000,C 90.000,E1 344.464} C_DIS
LIN {X -0.015,Y -195.310,Z 1191.891,A 0.000,B 0.000,C 90.000,E1 340.369} C_DIS
LIN {X -0.036,Y -200.648,Z 1191.868,A 0.000,B 0.000,C 90.000,E1 336.305} C_DIS
LIN {X -0.029,Y -206.622,Z 1191.846,A 0.000,B 0.000,C 90.000,E1 332.281} C_DIS
LIN {X -0.089,Y -213.152,Z 1191.824,A 0.000,B 0.000,C 90.000,E1 328.329} C_DIS
LIN {X -0.037,Y -220.285,Z 1191.802,A 0.000,B 0.000,C 90.000,E1 324.402} C_DIS
LIN {X 0.042,Y -226.518,Z 1191.785,A 0.000,B 0.000,C 90.000,E1 321.295} C_DIS
LIN {X 0.069,Y -233.545,Z 1191.768,A 0.000,B 0.000,C 90.000,E1 318.243} C_DIS
LIN {X 0.069,Y -241.642,Z 1191.751,A 0.000,B 0.000,C 90.000,E1 315.243} C_DIS
LIN {X -0.041,Y -251.061,Z 1191.735,A 0.000,B 0.000,C 90.000,E1 312.324} C_DIS
LIN {X -0.011,Y -262.851,Z 1191.717,A 0.000,B 0.000,C 90.000,E1 309.072} C_DIS
LIN {X 0.060,Y -272.860,Z 1191.703,A 0.000,B 0.000,C 90.000,E1 306.583} C_DIS
LIN {X -0.028,Y -280.710,Z 1191.694,A 0.000,B 0.000,C 90.000,E1 304.865} C_DIS
LIN {X -0.004,Y -296.390,Z 1191.677,A 0.000,B 0.000,C 90.000,E1 301.799} C_DIS
LIN {X 0.066,Y -308.141,Z 1191.666,A 0.000,B 0.000,C 90.000,E1 299.795} C_DIS
LIN {X -0.002,Y -318.807,Z 1191.657,A 0.000,B 0.000,C 90.000,E1 298.180} C_DIS
LIN {X 0.175,Y -328.026,Z 1191.649,A 0.000,B 0.000,C 90.000,E1 296.873} C_DIS
LIN {X -0.080,Y -338.183,Z 1191.643,A 0.000,B 0.000,C 90.000,E1 295.668} C_DIS
LIN {X -0.051,Y -359.513,Z 1191.629,A 0.000,B 0.000,C 90.000,E1 293.259} C_DIS
LIN {X -0.026,Y -383.788,Z 1191.615,A 0.000,B 0.000,C 90.000,E1 290.791} C_DIS
LIN {X -0.056,Y -397.288,Z 1191.608,A 0.000,B 0.000,C 90.000,E1 289.504} C_DIS
LIN {X 0.203,Y -410.410,Z 1191.601,A 0.000,B 0.000,C 90.000,E1 288.181} C_DIS
LIN {X -0.043,Y -420.610,Z 1191.595,A 0.000,B 0.000,C 90.000,E1 287.166} C_DIS
LIN {X 0.061,Y -427.663,Z 1191.591,A 0.000,B 0.000,C 90.000,E1 286.386} C_DIS
LIN {X -0.154,Y -434.689,Z 1191.587,A 0.000,B 0.000,C 90.000,E1 285.607} C_DIS
LIN {X 0.112,Y -441.141,Z 1191.582,A 0.000,B 0.000,C 90.000,E1 284.773} C_DIS
LIN {X -0.108,Y -446.845,Z 1191.578,A 0.000,B 0.000,C 90.000,E1 284.008} C_DIS
LIN {X -0.169,Y -451.925,Z 1191.573,A 0.000,B 0.000,C 90.000,E1 283.231} C_DIS
LIN {X 0.146,Y -456.364,Z 1191.569,A 0.000,B 0.000,C 90.000,E1 282.411} C_DIS
LIN {X -0.031,Y -459.987,Z 1191.565,A 0.000,B 0.000,C 90.000,E1 281.658} C_DIS
LIN {X -0.086,Y -463.018,Z 1191.560,A 0.000,B 0.000,C 90.000,E1 280.894} C_DIS
LIN {X 0.037,Y -464.652,Z 1191.558,A 0.000,B 0.000,C 90.000,E1 280.366} C_DIS
LIN {X 0.088,Y -465.997,Z 1191.555,A 0.000,B 0.000,C 90.000,E1 279.849} C_DIS
LIN {X -0.157,Y -468.169,Z 1191.549,A 0.000,B 0.000,C 90.000,E1 278.859} C_DIS
LIN {X -0.073,Y -469.059,Z 1191.546,A 0.000,B 0.000,C 90.000,E1 278.341} C_DIS
LIN {X 0.083,Y -469.744,Z 1191.543,A 0.000,B 0.000,C 90.000,E1 277.814} C_DIS
LIN {X 0.179,Y -470.091,Z 1191.541,A 0.000,B 0.000,C 90.000,E1 277.296} C_DIS
LIN {X -0.188,Y -470.046,Z 1191.538,A 0.000,B 0.000,C 90.000,E1 276.834} C_DIS
LIN {X -0.085,Y -469.559,Z 1191.535,A 0.000,B 0.000,C 90.000,E1 276.315} C_DIS
LIN {X 0.017,Y -468.636,Z 1191.532,A 0.000,B 0.000,C 90.000,E1 275.796} C_DIS
LIN {X 0.115,Y -467.242,Z 1191.529,A 0.000,B 0.000,C 90.000,E1 275.277} C_DIS
LIN {X 0.206,Y -465.361,Z 1191.527,A 0.000,B 0.000,C 90.000,E1 274.759} C_DIS
LIN {X -0.211,Y -462.967,Z 1191.524,A 0.000,B 0.000,C 90.000,E1 274.302} C_DIS
LIN {X -0.145,Y -459.896,Z 1191.521,A 0.000,B 0.000,C 90.000,E1 273.784} C_DIS
LIN {X -0.126,Y -456.047,Z 1191.518,A 0.000,B 0.000,C 90.000,E1 273.269} C_DIS
LIN {X -0.099,Y -451.113,Z 1191.515,A 0.000,B 0.000,C 90.000,E1 272.751} C_DIS
LIN {X 0.182,Y -448.186,Z 1191.514,A 0.000,B 0.000,C 90.000,E1 272.465} C_DIS
LIN {X 0.015,Y -444.897,Z 1191.512,A 0.000,B 0.000,C 90.000,E1 272.236} C_DIS
LIN {X 0.166,Y -441.719,Z 1191.511,A 0.000,B 0.000,C 90.000,E1 272.007} C_DIS
END
